Universal Robots PolyScope program: draw_test_name.urp

Program draw_test_name (installation=default directory=/programs createdIn=5.11.9.1010452 lastSavedIn=5.11.9.1010452 robotSerialNumber=20225200364)
Calibrated DH parameters: a=[0.00002, -0.569483, -0.54992, -0.00001, -0.000036, 0]; d=[0.180894, -146.691669, 192.918669, -46.053088, 0.119778, 0.115602]; alpha=[1.571425, -0.001534, 0.003359, 1.568739, -1.571477, 0]; deltaTheta=[0, 0.376258, -0.101074, -0.275185, -0.000002, 0]
Robot Program (runOnlyOnce=true)
  Script file /programs/usbdisk/draw_Marco_name.script
    | def Machining2():
    |   # Default parameters:
    |   global speed_ms = 0.3
    |   global speed_rads = 0.75
    |   global accel_mss = 3
    |   global accel_radss = 1.2
    |   global blend_radius_m = 0.001
    | 
    |   # Add subprograms here
    |   # Start of main program
    |   # Program generated by RoboDK v5.6.5 for UR10e on 20/10/2023 11:07:04
    |   # Using nominal kinematics.
    |   blend_radius_m = 0.001
    |   speed_ms = 1.000
    |   # set_reference(p[0.335000, -0.152000, -0.001000, 0.000000, 0.000000, 0.000000])
    |   set_tcp(p[0.000000, 0.000000, 0.252000, 0.000000, 0.000000, 0.000000])
    |   # Show Tool
    |   movej([0.142122, -1.120207, -2.573393, -1.018789, 1.570796, 1.712919],accel_radss,speed_rads,0,blend_radius_m)
    |   movel([0.142122, -1.120207, -2.573393, -1.018789, 1.570796, 1.712919],accel_mss,speed_ms,0,blend_radius_m)
    |   # Splitting Linear movement in 72 (instruction 7: MoveL 3)
    |   movel([0.142122, -1.121315, -2.574321, -1.016753, 1.570796, 1.712919],accel_mss,speed_ms,0,blend_radius_m)
    |   movel([0.142122, -1.122427, -2.575248, -1.014714, 1.570796, 1.712919],accel_mss,speed_ms,0,blend_radius_m)
    |   movel([0.142122, -1.123545, -2.576174, -1.012670, 1.570796, 1.712919],accel_mss,speed_ms,0,blend_radius_m)
    |   movel([0.142122, -1.124668, -2.577098, -1.010623, 1.570796, 1.712919],accel_mss,speed_ms,0,blend_radius_m)
    |   movel([0.142122, -1.125797, -2.578021, -1.008571, 1.570796, 1.712919],accel_mss,speed_ms,0,blend_radius_m)
    |   movel([0.142122, -1.126931, -2.578943, -1.006515, 1.570796, 1.712919],accel_mss,speed_ms,0,blend_radius_m)
    |   movel([0.142122, -1.128070, -2.579864, -1.004456, 1.570796, 1.712919],accel_mss,speed_ms,0,blend_radius_m)
    |   movel([0.142122, -1.129214, -2.580783, -1.002392, 1.570796, 1.712919],accel_mss,speed_ms,0,blend_radius_m)
    |   movel([0.142122, -1.130364, -2.581701, -1.000323, 1.570796, 1.712919],accel_mss,speed_ms,0,blend_radius_m)
    |   movel([0.142122, -1.131520, -2.582618, -0.998251, 1.570796, 1.712919],accel_mss,speed_ms,0,blend_radius_m)
    |   movel([0.142122, -1.132681, -2.583534, -0.996175, 1.570796, 1.712919],accel_mss,speed_ms,0,blend_radius_m)
    |   movel([0.142122, -1.133847, -2.584448, -0.994094, 1.570796, 1.712919],accel_mss,speed_ms,0,blend_radius_m)
    |   movel([0.142122, -1.135018, -2.585361, -0.992009, 1.570796, 1.712919],accel_mss,speed_ms,0,blend_radius_m)
    |   movel([0.142122, -1.136196, -2.586273, -0.989920, 1.570796, 1.712919],accel_mss,speed_ms,0,blend_radius_m)
    |   movel([0.142122, -1.137378, -2.587184, -0.987827, 1.570796, 1.712919],accel_mss,speed_ms,0,blend_radius_m)
    |   movel([0.142122, -1.138567, -2.588093, -0.985729, 1.570796, 1.712919],accel_mss,speed_ms,0,blend_radius_m)
    |   movel([0.142122, -1.139760, -2.589001, -0.983628, 1.570796, 1.712919],accel_mss,speed_ms,0,blend_radius_m)
    |   movel([0.142122, -1.140959, -2.589908, -0.981522, 1.570796, 1.712919],accel_mss,speed_ms,0,blend_radius_m)
    |   movel([0.142122, -1.142164, -2.590813, -0.979411, 1.570796, 1.712919],accel_mss,speed_ms,0,blend_radius_m)
    |   movel([0.142122, -1.143375, -2.591717, -0.977297, 1.570796, 1.712919],accel_mss,speed_ms,0,blend_radius_m)
    |   movel([0.142122, -1.144591, -2.592620, -0.975178, 1.570796, 1.712919],accel_mss,speed_ms,0,blend_radius_m)
    |   movel([0.142122, -1.145812, -2.593522, -0.973055, 1.570796, 1.712919],accel_mss,speed_ms,0,blend_radius_m)
    |   movel([0.142122, -1.147039, -2.594422, -0.970928, 1.570796, 1.712919],accel_mss,speed_ms,0,blend_radius_m)
    |   movel([0.142122, -1.148272, -2.595321, -0.968796, 1.570796, 1.712919],accel_mss,speed_ms,0,blend_radius_m)
    |   movel([0.142122, -1.149511, -2.596218, -0.966660, 1.570796, 1.712919],accel_mss,speed_ms,0,blend_radius_m)
    |   movel([0.142122, -1.150755, -2.597115, -0.964519, 1.570796, 1.712919],accel_mss,speed_ms,0,blend_radius_m)
    |   movel([0.142122, -1.152005, -2.598010, -0.962374, 1.570796, 1.712919],accel_mss,speed_ms,0,blend_radius_m)
    |   movel([0.142122, -1.153261, -2.598903, -0.960225, 1.570796, 1.712919],accel_mss,speed_ms,0,blend_radius_m)
    |   movel([0.142122, -1.154522, -2.599795, -0.958072, 1.570796, 1.712919],accel_mss,speed_ms,0,blend_radius_m)
    |   movel([0.142122, -1.155789, -2.600686, -0.955914, 1.570796, 1.712919],accel_mss,speed_ms,0,blend_radius_m)
    |   movel([0.142122, -1.157062, -2.601576, -0.953751, 1.570796, 1.712919],accel_mss,speed_ms,0,blend_radius_m)
    |   movel([0.142122, -1.158341, -2.602464, -0.951585, 1.570796, 1.712919],accel_mss,speed_ms,0,blend_radius_m)
    |   movel([0.142122, -1.159625, -2.603351, -0.949413, 1.570796, 1.712919],accel_mss,speed_ms,0,blend_radius_m)
    |   movel([0.142122, -1.160915, -2.604236, -0.947238, 1.570796, 1.712919],accel_mss,speed_ms,0,blend_radius_m)
    |   movel([0.142122, -1.162211, -2.605120, -0.945058, 1.570796, 1.712919],accel_mss,speed_ms,0,blend_radius_m)
    |   movel([0.142122, -1.163513, -2.606003, -0.942873, 1.570796, 1.712919],accel_mss,speed_ms,0,blend_radius_m)
    |   movel([0.142122, -1.164821, -2.606884, -0.940684, 1.570796, 1.712919],accel_mss,speed_ms,0,blend_radius_m)
    |   movel([0.142122, -1.166135, -2.607764, -0.938490, 1.570796, 1.712919],accel_mss,speed_ms,0,blend_radius_m)
    |   movel([0.142122, -1.167455, -2.608642, -0.936292, 1.570796, 1.712919],accel_mss,speed_ms,0,blend_radius_m)
    |   movel([0.142122, -1.168780, -2.609519, -0.934090, 1.570796, 1.712919],accel_mss,speed_ms,0,blend_radius_m)
    |   movel([0.142122, -1.170112, -2.610395, -0.931882, 1.570796, 1.712919],accel_mss,speed_ms,0,blend_radius_m)
    |   movel([0.142122, -1.171449, -2.611269, -0.929671, 1.570796, 1.712919],accel_mss,speed_ms,0,blend_radius_m)
    |   movel([0.142122, -1.172792, -2.612142, -0.927455, 1.570796, 1.712919],accel_mss,speed_ms,0,blend_radius_m)
    |   movel([0.142122, -1.174142, -2.613013, -0.925234, 1.570796, 1.712919],accel_mss,speed_ms,0,blend_radius_m)
    |   movel([0.142122, -1.175497, -2.613883, -0.923008, 1.570796, 1.712919],accel_mss,speed_ms,0,blend_radius_m)
    |   movel([0.142122, -1.176859, -2.614752, -0.920779, 1.570796, 1.712919],accel_mss,speed_ms,0,blend_radius_m)
    |   movel([0.142122, -1.178226, -2.615619, -0.918544, 1.570796, 1.712919],accel_mss,speed_ms,0,blend_radius_m)
    |   movel([0.142122, -1.179600, -2.616484, -0.916305, 1.570796, 1.712919],accel_mss,speed_ms,0,blend_radius_m)
    |   movel([0.142122, -1.180979, -2.617348, -0.914061, 1.570796, 1.712919],accel_mss,speed_ms,0,blend_radius_m)
    |   movel([0.142122, -1.182365, -2.618211, -0.911813, 1.570796, 1.712919],accel_mss,speed_ms,0,blend_radius_m)
    |   movel([0.142122, -1.183757, -2.619072, -0.909560, 1.570796, 1.712919],accel_mss,speed_ms,0,blend_radius_m)
    |   movel([0.142122, -1.185155, -2.619932, -0.907302, 1.570796, 1.712919],accel_mss,speed_ms,0,blend_radius_m)
    |   movel([0.142122, -1.186559, -2.620790, -0.905040, 1.570796, 1.712919],accel_mss,speed_ms,0,blend_radius_m)
    |   movel([0.142122, -1.187969, -2.621647, -0.902773, 1.570796, 1.712919],accel_mss,speed_ms,0,blend_radius_m)
    |   movel([0.142122, -1.189386, -2.622502, -0.900501, 1.570796, 1.712919],accel_mss,speed_ms,0,blend_radius_m)
    |   movel([0.142122, -1.190808, -2.623356, -0.898225, 1.570796, 1.712919],accel_mss,speed_ms,0,blend_radius_m)
    |   movel([0.142122, -1.192237, -2.624208, -0.895943, 1.570796, 1.712919],accel_mss,speed_ms,0,blend_radius_m)
    |   movel([0.142122, -1.193672, -2.625059, -0.893658, 1.570796, 1.712919],accel_mss,speed_ms,0,blend_radius_m)
    |   movel([0.142122, -1.195113, -2.625908, -0.891367, 1.570796, 1.712919],accel_mss,speed_ms,0,blend_radius_m)
    |   movel([0.142122, -1.196561, -2.626756, -0.889072, 1.570796, 1.712919],accel_mss,speed_ms,0,blend_radius_m)
    |   movel([0.142122, -1.198015, -2.627602, -0.886772, 1.570796, 1.712919],accel_mss,speed_ms,0,blend_radius_m)
    |   movel([0.142122, -1.199475, -2.628447, -0.884467, 1.570796, 1.712919],accel_mss,speed_ms,0,blend_radius_m)
    |   movel([0.142122, -1.200942, -2.629290, -0.882157, 1.570796, 1.712919],accel_mss,speed_ms,0,blend_radius_m)
    |   movel([0.142122, -1.202414, -2.630132, -0.879843, 1.570796, 1.712919],accel_mss,speed_ms,0,blend_radius_m)
    |   movel([0.142122, -1.203893, -2.630972, -0.877524, 1.570796, 1.712919],accel_mss,speed_ms,0,blend_radius_m)
    |   movel([0.142122, -1.205379, -2.631810, -0.875200, 1.570796, 1.712919],accel_mss,speed_ms,0,blend_radius_m)
    |   movel([0.142122, -1.206871, -2.632647, -0.872871, 1.570796, 1.712919],accel_mss,speed_ms,0,blend_radius_m)
    |   movel([0.142122, -1.208369, -2.633482, -0.870538, 1.570796, 1.712919],accel_mss,speed_ms,0,blend_radius_m)
    |   movel([0.142122, -1.209874, -2.634316, -0.868199, 1.570796, 1.712919],accel_mss,speed_ms,0,blend_radius_m)
    |   movel([0.142122, -1.211385, -2.635148, -0.865856, 1.570796, 1.712919],accel_mss,speed_ms,0,blend_radius_m)
    |   movel([0.142122, -1.212902, -2.635979, -0.863508, 1.570796, 1.712919],accel_mss,speed_ms,0,blend_radius_m)
    |   movel([0.142122, -1.214426, -2.636807, -0.861155, 1.570796, 1.712919],accel_mss,speed_ms,0,blend_radius_m)
    |   movel([0.142122, -1.214426, -2.636807, -0.861155, 1.570796, 1.712919],accel_mss,speed_ms,0,blend_radius_m)
    |   speed_ms = 1.000
    |   # Splitting Linear movement in 8 (instruction 10: MoveL 5)
    |   movel([0.142122, -1.215804, -2.637552, -0.859033, 1.570796, 1.712919],accel_mss,speed_ms,0,blend_radius_m)
    |   movel([0.142122, -1.217186, -2.638295, -0.856907, 1.570796, 1.712919],accel_mss,speed_ms,0,blend_radius_m)
    |   movel([0.142122, -1.218574, -2.639038, -0.854778, 1.570796, 1.712919],accel_mss,speed_ms,0,blend_radius_m)
    |   movel([0.142122, -1.219967, -2.639778, -0.852644, 1.570796, 1.712919],accel_mss,speed_ms,0,blend_radius_m)
    |   movel([0.142122, -1.221365, -2.640518, -0.850506, 1.570796, 1.712919],accel_mss,speed_ms,0,blend_radius_m)
    |   movel([0.142122, -1.222769, -2.641256, -0.848365, 1.570796, 1.712919],accel_mss,speed_ms,0,blend_radius_m)
    |   movel([0.142122, -1.224177, -2.641992, -0.846219, 1.570796, 1.712919],accel_mss,speed_ms,0,blend_radius_m)
    |   movel([0.142122, -1.225592, -2.642728, -0.844069, 1.570796, 1.712919],accel_mss,speed_ms,0,blend_radius_m)
    |   movel([0.142122, -1.225592, -2.642728, -0.844069, 1.570796, 1.712919],accel_mss,speed_ms,0,blend_radius_m)
    |   # Splitting Linear movement in 16 (instruction 12: MoveL 7)
    |   movel([0.142122, -1.227011, -2.643462, -0.841916, 1.570796, 1.712919],accel_mss,speed_ms,0,blend_radius_m)
    |   movel([0.142122, -1.228436, -2.644195, -0.839758, 1.570796, 1.712919],accel_mss,speed_ms,0,blend_radius_m)
    |   movel([0.142122, -1.229866, -2.644926, -0.837597, 1.570796, 1.712919],accel_mss,speed_ms,0,blend_radius_m)
    |   movel([0.142122, -1.231302, -2.645656, -0.835431, 1.570796, 1.712919],accel_mss,speed_ms,0,blend_radius_m)
    |   movel([0.142122, -1.232743, -2.646385, -0.833261, 1.570796, 1.712919],accel_mss,speed_ms,0,blend_radius_m)
    |   movel([0.142122, -1.234189, -2.647112, -0.831088, 1.570796, 1.712919],accel_mss,speed_ms,0,blend_radius_m)
    |   movel([0.142122, -1.235641, -2.647838, -0.828910, 1.570796, 1.712919],accel_mss,speed_ms,0,blend_radius_m)
    |   movel([0.142122, -1.237099, -2.648562, -0.826728, 1.570796, 1.712919],accel_mss,speed_ms,0,blend_radius_m)
    |   movel([0.142122, -1.238561, -2.649286, -0.824542, 1.570796, 1.712919],accel_mss,speed_ms,0,blend_radius_m)
    |   movel([0.142122, -1.240029, -2.650007, -0.822352, 1.570796, 1.712919],accel_mss,speed_ms,0,blend_radius_m)
    |   movel([0.142122, -1.241503, -2.650728, -0.820158, 1.570796, 1.712919],accel_mss,speed_ms,0,blend_radius_m)
    |   movel([0.142122, -1.242982, -2.651447, -0.817960, 1.570796, 1.712919],accel_mss,speed_ms,0,blend_radius_m)
    |   movel([0.142122, -1.244466, -2.652164, -0.815758, 1.570796, 1.712919],accel_mss,speed_ms,0,blend_radius_m)
    |   movel([0.142122, -1.245956, -2.652880, -0.813552, 1.570796, 1.712919],accel_mss,speed_ms,0,blend_radius_m)
    |   movel([0.142122, -1.247452, -2.653595, -0.811342, 1.570796, 1.712919],accel_mss,speed_ms,0,blend_radius_m)
    |   movel([0.142122, -1.248953, -2.654308, -0.809128, 1.570796, 1.712919],accel_mss,speed_ms,0,blend_radius_m)
    |   # Splitting Linear movement in 6 (instruction 13: MoveL 8)
    |   movel([0.140118, -1.249589, -2.653970, -0.808830, 1.570796, 1.710915],accel_mss,speed_ms,0,blend_radius_m)
    |   movel([0.138115, -1.250228, -2.653630, -0.808531, 1.570796, 1.708912],accel_mss,speed_ms,0,blend_radius_m)
    |   movel([0.136113, -1.250869, -2.653288, -0.808232, 1.570796, 1.706910],accel_mss,speed_ms,0,blend_radius_m)
    |   movel([0.134112, -1.251512, -2.652944, -0.807932, 1.570796, 1.704909],accel_mss,speed_ms,0,blend_radius_m)
    |   movel([0.132112, -1.252158, -2.652599, -0.807632, 1.570796, 1.702908],accel_mss,speed_ms,0,blend_radius_m)
    |   movel([0.130113, -1.252807, -2.652252, -0.807331, 1.570796, 1.700909],accel_mss,speed_ms,0,blend_radius_m)
    |   # Splitting Linear movement in 16 (instruction 14: MoveL 9)
    |   movel([0.130113, -1.251309, -2.651541, -0.809539, 1.570796, 1.700909],accel_mss,speed_ms,0,blend_radius_m)
    |   movel([0.130113, -1.249816, -2.650829, -0.811744, 1.570796, 1.700909],accel_mss,speed_ms,0,blend_radius_m)
    |   movel([0.130113, -1.248329, -2.650116, -0.813944, 1.570796, 1.700909],accel_mss,speed_ms,0,blend_radius_m)
    |   movel([0.130113, -1.246847, -2.649401, -0.816141, 1.570796, 1.700909],accel_mss,speed_ms,0,blend_radius_m)
    |   movel([0.130113, -1.245371, -2.648685, -0.818333, 1.570796, 1.700909],accel_mss,speed_ms,0,blend_radius_m)
    |   movel([0.130113, -1.243900, -2.647967, -0.820522, 1.570796, 1.700909],accel_mss,speed_ms,0,blend_radius_m)
    |   movel([0.130113, -1.242435, -2.647248, -0.822706, 1.570796, 1.700909],accel_mss,speed_ms,0,blend_radius_m)
    |   movel([0.130113, -1.240974, -2.646528, -0.824887, 1.570796, 1.700909],accel_mss,speed_ms,0,blend_radius_m)
    |   movel([0.130113, -1.239520, -2.645806, -0.827063, 1.570796, 1.700909],accel_mss,speed_ms,0,blend_radius_m)
    |   movel([0.130113, -1.238071, -2.645083, -0.829236, 1.570796, 1.700909],accel_mss,speed_ms,0,blend_radius_m)
    |   movel([0.130113, -1.236627, -2.644358, -0.831404, 1.570796, 1.700909],accel_mss,speed_ms,0,blend_radius_m)
    |   movel([0.130113, -1.235188, -2.643632, -0.833569, 1.570796, 1.700909],accel_mss,speed_ms,0,blend_radius_m)
    |   movel([0.130113, -1.233755, -2.642905, -0.835729, 1.570796, 1.700909],accel_mss,speed_ms,0,blend_radius_m)
    |   movel([0.130113, -1.232327, -2.642176, -0.837886, 1.570796, 1.700909],accel_mss,speed_ms,0,blend_radius_m)
    |   movel([0.130113, -1.230904, -2.641446, -0.840038, 1.570796, 1.700909],accel_mss,speed_ms,0,blend_radius_m)
    |   movel([0.130113, -1.229487, -2.640715, -0.842187, 1.570796, 1.700909],accel_mss,speed_ms,0,blend_radius_m)
    |   # Splitting Linear movement in 6 (instruction 15: MoveL 10)
    |   movel([0.132112, -1.228832, -2.641055, -0.842503, 1.570796, 1.702908],accel_mss,speed_ms,0,blend_radius_m)
    |   movel([0.134112, -1.228179, -2.641393, -0.842817, 1.570796, 1.704909],accel_mss,speed_ms,0,blend_radius_m)
    |   movel([0.136113, -1.227528, -2.641729, -0.843131, 1.570796, 1.706910],accel_mss,speed_ms,0,blend_radius_m)
    |   movel([0.138115, -1.226880, -2.642064, -0.843445, 1.570796, 1.708912],accel_mss,speed_ms,0,blend_radius_m)
    |   movel([0.140118, -1.226235, -2.642397, -0.843758, 1.570796, 1.710915],accel_mss,speed_ms,0,blend_radius_m)
    |   movel([0.142122, -1.225592, -2.642728, -0.844069, 1.570796, 1.712919],accel_mss,speed_ms,0,blend_radius_m)
    |   # Splitting Linear movement in 16 (instruction 16: MoveL 11)
    |   movel([0.142122, -1.227011, -2.643462, -0.841916, 1.570796, 1.712919],accel_mss,speed_ms,0,blend_radius_m)
    |   movel([0.142122, -1.228436, -2.644195, -0.839758, 1.570796, 1.712919],accel_mss,speed_ms,0,blend_radius_m)
    |   movel([0.142122, -1.229866, -2.644926, -0.837597, 1.570796, 1.712919],accel_mss,speed_ms,0,blend_radius_m)
    |   movel([0.142122, -1.231302, -2.645656, -0.835431, 1.570796, 1.712919],accel_mss,speed_ms,0,blend_radius_m)
    |   movel([0.142122, -1.232743, -2.646385, -0.833261, 1.570796, 1.712919],accel_mss,speed_ms,0,blend_radius_m)
    |   movel([0.142122, -1.234189, -2.647112, -0.831088, 1.570796, 1.712919],accel_mss,speed_ms,0,blend_radius_m)
    |   movel([0.142122, -1.235641, -2.647838, -0.828910, 1.570796, 1.712919],accel_mss,speed_ms,0,blend_radius_m)
    |   movel([0.142122, -1.237099, -2.648562, -0.826728, 1.570796, 1.712919],accel_mss,speed_ms,0,blend_radius_m)
    |   movel([0.142122, -1.238561, -2.649286, -0.824542, 1.570796, 1.712919],accel_mss,speed_ms,0,blend_radius_m)
    |   movel([0.142122, -1.240029, -2.650007, -0.822352, 1.570796, 1.712919],accel_mss,speed_ms,0,blend_radius_m)
    |   movel([0.142122, -1.241503, -2.650728, -0.820158, 1.570796, 1.712919],accel_mss,speed_ms,0,blend_radius_m)
    |   movel([0.142122, -1.242982, -2.651447, -0.817960, 1.570796, 1.712919],accel_mss,speed_ms,0,blend_radius_m)
    |   movel([0.142122, -1.244466, -2.652164, -0.815758, 1.570796, 1.712919],accel_mss,speed_ms,0,blend_radius_m)
    |   movel([0.142122, -1.245956, -2.652880, -0.813552, 1.570796, 1.712919],accel_mss,speed_ms,0,blend_radius_m)
    |   movel([0.142122, -1.247452, -2.653595, -0.811342, 1.570796, 1.712919],accel_mss,speed_ms,0,blend_radius_m)
    |   movel([0.142122, -1.248953, -2.654308, -0.809128, 1.570796, 1.712919],accel_mss,speed_ms,0,blend_radius_m)
    |   # Splitting Linear movement in 8 (instruction 17: MoveL 12)
    |   movel([0.140538, -1.249956, -2.653775, -0.808658, 1.570796, 1.711335],accel_mss,speed_ms,0,blend_radius_m)
    |   movel([0.138957, -1.250958, -2.653241, -0.808191, 1.570796, 1.709753],accel_mss,speed_ms,0,blend_radius_m)
    |   movel([0.137378, -1.251960, -2.652705, -0.807724, 1.570796, 1.708174],accel_mss,speed_ms,0,blend_radius_m)
    |   movel([0.135801, -1.252961, -2.652169, -0.807259, 1.570796, 1.706597],accel_mss,speed_ms,0,blend_radius_m)
    |   movel([0.134226, -1.253962, -2.651632, -0.806795, 1.570796, 1.705023],accel_mss,speed_ms,0,blend_radius_m)
    |   movel([0.132655, -1.254963, -2.651093, -0.806333, 1.570796, 1.703451],accel_mss,speed_ms,0,blend_radius_m)
    |   movel([0.131085, -1.255963, -2.650554, -0.805872, 1.570796, 1.701881],accel_mss,speed_ms,0,blend_radius_m)
    |   movel([0.129518, -1.256963, -2.650014, -0.805412, 1.570796, 1.700314],accel_mss,speed_ms,0,blend_radius_m)
    |   # Splitting Linear movement in 16 (instruction 18: MoveL 13)
    |   movel([0.129518, -1.255469, -2.649306, -0.807614, 1.570796, 1.700314],accel_mss,speed_ms,0,blend_radius_m)
    |   movel([0.129518, -1.253979, -2.648597, -0.809813, 1.570796, 1.700314],accel_mss,speed_ms,0,blend_radius_m)
    |   movel([0.129518, -1.252495, -2.647887, -0.812007, 1.570796, 1.700314],accel_mss,speed_ms,0,blend_radius_m)
    |   movel([0.129518, -1.251017, -2.647175, -0.814198, 1.570796, 1.700314],accel_mss,speed_ms,0,blend_radius_m)
    |   movel([0.129518, -1.249543, -2.646461, -0.816384, 1.570796, 1.700314],accel_mss,speed_ms,0,blend_radius_m)
    |   movel([0.129518, -1.248076, -2.645747, -0.818567, 1.570796, 1.700314],accel_mss,speed_ms,0,blend_radius_m)
    |   movel([0.129518, -1.246613, -2.645031, -0.820745, 1.570796, 1.700314],accel_mss,speed_ms,0,blend_radius_m)
    |   movel([0.129518, -1.245156, -2.644313, -0.822920, 1.570796, 1.700314],accel_mss,speed_ms,0,blend_radius_m)
    |   movel([0.129518, -1.243704, -2.643594, -0.825091, 1.570796, 1.700314],accel_mss,speed_ms,0,blend_radius_m)
    |   movel([0.129518, -1.242257, -2.642874, -0.827257, 1.570796, 1.700314],accel_mss,speed_ms,0,blend_radius_m)
    |   movel([0.129518, -1.240816, -2.642152, -0.829420, 1.570796, 1.700314],accel_mss,speed_ms,0,blend_radius_m)
    |   movel([0.129518, -1.239380, -2.641429, -0.831579, 1.570796, 1.700314],accel_mss,speed_ms,0,blend_radius_m)
    |   movel([0.129518, -1.237950, -2.640705, -0.833734, 1.570796, 1.700314],accel_mss,speed_ms,0,blend_radius_m)
    |   movel([0.129518, -1.236524, -2.639979, -0.835885, 1.570796, 1.700314],accel_mss,speed_ms,0,blend_radius_m)
    |   movel([0.129518, -1.235104, -2.639252, -0.838032, 1.570796, 1.700314],accel_mss,speed_ms,0,blend_radius_m)
    |   movel([0.129518, -1.233690, -2.638524, -0.840176, 1.570796, 1.700314],accel_mss,speed_ms,0,blend_radius_m)
    |   # Splitting Linear movement in 8 (instruction 19: MoveL 14)
    |   movel([0.130935, -1.233727, -2.638504, -0.840158, 1.570796, 1.701732],accel_mss,speed_ms,0,blend_radius_m)
    |   movel([0.132351, -1.233767, -2.638483, -0.840139, 1.570796, 1.703148],accel_mss,speed_ms,0,blend_radius_m)
    |   movel([0.133766, -1.233809, -2.638461, -0.840119, 1.570796, 1.704563],accel_mss,speed_ms,0,blend_radius_m)
    |   movel([0.135180, -1.233853, -2.638438, -0.840098, 1.570796, 1.705976],accel_mss,speed_ms,0,blend_radius_m)
    |   movel([0.136593, -1.233900, -2.638414, -0.840075, 1.570796, 1.707389],accel_mss,speed_ms,0,blend_radius_m)
    |   movel([0.138004, -1.233949, -2.638388, -0.840052, 1.570796, 1.708800],accel_mss,speed_ms,0,blend_radius_m)
    |   movel([0.139414, -1.234000, -2.638361, -0.840028, 1.570796, 1.710211],accel_mss,speed_ms,0,blend_radius_m)
    |   movel([0.140824, -1.234053, -2.638333, -0.840003, 1.570796, 1.711620],accel_mss,speed_ms,0,blend_radius_m)
    |   # Splitting Linear movement in 16 (instruction 20: MoveL 15)
    |   movel([0.140824, -1.235468, -2.639062, -0.837860, 1.570796, 1.711620],accel_mss,speed_ms,0,blend_radius_m)
    |   movel([0.140824, -1.236888, -2.639788, -0.835713, 1.570796, 1.711620],accel_mss,speed_ms,0,blend_radius_m)
    |   movel([0.140824, -1.238313, -2.640514, -0.833563, 1.570796, 1.711620],accel_mss,speed_ms,0,blend_radius_m)
    |   movel([0.140824, -1.239743, -2.641238, -0.831408, 1.570796, 1.711620],accel_mss,speed_ms,0,blend_radius_m)
    |   movel([0.140824, -1.241179, -2.641961, -0.829250, 1.570796, 1.711620],accel_mss,speed_ms,0,blend_radius_m)
    |   movel([0.140824, -1.242620, -2.642682, -0.827087, 1.570796, 1.711620],accel_mss,speed_ms,0,blend_radius_m)
    |   movel([0.140824, -1.244066, -2.643402, -0.824921, 1.570796, 1.711620],accel_mss,speed_ms,0,blend_radius_m)
    |   movel([0.140824, -1.245518, -2.644121, -0.822751, 1.570796, 1.711620],accel_mss,speed_ms,0,blend_radius_m)
    |   movel([0.140824, -1.246974, -2.644838, -0.820577, 1.570796, 1.711620],accel_mss,speed_ms,0,blend_radius_m)
    |   movel([0.140824, -1.248437, -2.645554, -0.818399, 1.570796, 1.711620],accel_mss,speed_ms,0,blend_radius_m)
    |   movel([0.140824, -1.249904, -2.646268, -0.816217, 1.570796, 1.711620],accel_mss,speed_ms,0,blend_radius_m)
    |   movel([0.140824, -1.251377, -2.646981, -0.814031, 1.570796, 1.711620],accel_mss,speed_ms,0,blend_radius_m)
    |   movel([0.140824, -1.252856, -2.647693, -0.811841, 1.570796, 1.711620],accel_mss,speed_ms,0,blend_radius_m)
    |   movel([0.140824, -1.254339, -2.648403, -0.809647, 1.570796, 1.711620],accel_mss,speed_ms,0,blend_radius_m)
    |   movel([0.140824, -1.255828, -2.649112, -0.807449, 1.570796, 1.711620],accel_mss,speed_ms,0,blend_radius_m)
    |   movel([0.140824, -1.257323, -2.649819, -0.805247, 1.570796, 1.711620],accel_mss,speed_ms,0,blend_radius_m)
    |   # Splitting Linear movement in 8 (instruction 21: MoveL 16)
    |   movel([0.139414, -1.257270, -2.649847, -0.805271, 1.570796, 1.710211],accel_mss,speed_ms,0,blend_radius_m)
    |   movel([0.138004, -1.257220, -2.649875, -0.805294, 1.570796, 1.708800],accel_mss,speed_ms,0,blend_radius_m)
    |   movel([0.136593, -1.257171, -2.649901, -0.805317, 1.570796, 1.707389],accel_mss,speed_ms,0,blend_radius_m)
    |   movel([0.135180, -1.257125, -2.649926, -0.805338, 1.570796, 1.705976],accel_mss,speed_ms,0,blend_radius_m)
    |   movel([0.133766, -1.257082, -2.649950, -0.805358, 1.570796, 1.704563],accel_mss,speed_ms,0,blend_radius_m)
    |   movel([0.132351, -1.257040, -2.649972, -0.805377, 1.570796, 1.703148],accel_mss,speed_ms,0,blend_radius_m)
    |   movel([0.130935, -1.257001, -2.649993, -0.805395, 1.570796, 1.701732],accel_mss,speed_ms,0,blend_radius_m)
    |   movel([0.129518, -1.256963, -2.650014, -0.805412, 1.570796, 1.700314],accel_mss,speed_ms,0,blend_radius_m)
    |   # Splitting Linear movement in 16 (instruction 22: MoveL 17)
    |   movel([0.129518, -1.255469, -2.649306, -0.807614, 1.570796, 1.700314],accel_mss,speed_ms,0,blend_radius_m)
    |   movel([0.129518, -1.253979, -2.648597, -0.809813, 1.570796, 1.700314],accel_mss,speed_ms,0,blend_radius_m)
    |   movel([0.129518, -1.252495, -2.647887, -0.812007, 1.570796, 1.700314],accel_mss,speed_ms,0,blend_radius_m)
    |   movel([0.129518, -1.251017, -2.647175, -0.814198, 1.570796, 1.700314],accel_mss,speed_ms,0,blend_radius_m)
    |   movel([0.129518, -1.249543, -2.646461, -0.816384, 1.570796, 1.700314],accel_mss,speed_ms,0,blend_radius_m)
    |   movel([0.129518, -1.248076, -2.645747, -0.818567, 1.570796, 1.700314],accel_mss,speed_ms,0,blend_radius_m)
    |   movel([0.129518, -1.246613, -2.645031, -0.820745, 1.570796, 1.700314],accel_mss,speed_ms,0,blend_radius_m)
    |   movel([0.129518, -1.245156, -2.644313, -0.822920, 1.570796, 1.700314],accel_mss,speed_ms,0,blend_radius_m)
    |   movel([0.129518, -1.243704, -2.643594, -0.825091, 1.570796, 1.700314],accel_mss,speed_ms,0,blend_radius_m)
    |   movel([0.129518, -1.242257, -2.642874, -0.827257, 1.570796, 1.700314],accel_mss,speed_ms,0,blend_radius_m)
    |   movel([0.129518, -1.240816, -2.642152, -0.829420, 1.570796, 1.700314],accel_mss,speed_ms,0,blend_radius_m)
    |   movel([0.129518, -1.239380, -2.641429, -0.831579, 1.570796, 1.700314],accel_mss,speed_ms,0,blend_radius_m)
    |   movel([0.129518, -1.237950, -2.640705, -0.833734, 1.570796, 1.700314],accel_mss,speed_ms,0,blend_radius_m)
    |   movel([0.129518, -1.236524, -2.639979, -0.835885, 1.570796, 1.700314],accel_mss,speed_ms,0,blend_radius_m)
    |   movel([0.129518, -1.235104, -2.639252, -0.838032, 1.570796, 1.700314],accel_mss,speed_ms,0,blend_radius_m)
    |   movel([0.129518, -1.233690, -2.638524, -0.840176, 1.570796, 1.700314],accel_mss,speed_ms,0,blend_radius_m)
    |   # Splitting Linear movement in 8 (instruction 23: MoveL 18)
    |   movel([0.130935, -1.233727, -2.638504, -0.840158, 1.570796, 1.701732],accel_mss,speed_ms,0,blend_radius_m)
    |   movel([0.132351, -1.233767, -2.638483, -0.840139, 1.570796, 1.703148],accel_mss,speed_ms,0,blend_radius_m)
    |   movel([0.133766, -1.233809, -2.638461, -0.840119, 1.570796, 1.704563],accel_mss,speed_ms,0,blend_radius_m)
    |   movel([0.135180, -1.233853, -2.638438, -0.840098, 1.570796, 1.705976],accel_mss,speed_ms,0,blend_radius_m)
    |   movel([0.136593, -1.233900, -2.638414, -0.840075, 1.570796, 1.707389],accel_mss,speed_ms,0,blend_radius_m)
    |   movel([0.138004, -1.233949, -2.638388, -0.840052, 1.570796, 1.708800],accel_mss,speed_ms,0,blend_radius_m)
    |   movel([0.139414, -1.234000, -2.638361, -0.840028, 1.570796, 1.710211],accel_mss,speed_ms,0,blend_radius_m)
    |   movel([0.140824, -1.234053, -2.638333, -0.840003, 1.570796, 1.711620],accel_mss,speed_ms,0,blend_radius_m)
    |   # Splitting Linear movement in 16 (instruction 24: MoveL 19)
    |   movel([0.140824, -1.235468, -2.639062, -0.837860, 1.570796, 1.711620],accel_mss,speed_ms,0,blend_radius_m)
    |   movel([0.140824, -1.236888, -2.639788, -0.835713, 1.570796, 1.711620],accel_mss,speed_ms,0,blend_radius_m)
    |   movel([0.140824, -1.238313, -2.640514, -0.833563, 1.570796, 1.711620],accel_mss,speed_ms,0,blend_radius_m)
    |   movel([0.140824, -1.239743, -2.641238, -0.831408, 1.570796, 1.711620],accel_mss,speed_ms,0,blend_radius_m)
    |   movel([0.140824, -1.241179, -2.641961, -0.829250, 1.570796, 1.711620],accel_mss,speed_ms,0,blend_radius_m)
    |   movel([0.140824, -1.242620, -2.642682, -0.827087, 1.570796, 1.711620],accel_mss,speed_ms,0,blend_radius_m)
    |   movel([0.140824, -1.244066, -2.643402, -0.824921, 1.570796, 1.711620],accel_mss,speed_ms,0,blend_radius_m)
    |   movel([0.140824, -1.245518, -2.644121, -0.822751, 1.570796, 1.711620],accel_mss,speed_ms,0,blend_radius_m)
    |   movel([0.140824, -1.246974, -2.644838, -0.820577, 1.570796, 1.711620],accel_mss,speed_ms,0,blend_radius_m)
    |   movel([0.140824, -1.248437, -2.645554, -0.818399, 1.570796, 1.711620],accel_mss,speed_ms,0,blend_radius_m)
    |   movel([0.140824, -1.249904, -2.646268, -0.816217, 1.570796, 1.711620],accel_mss,speed_ms,0,blend_radius_m)
    |   movel([0.140824, -1.251377, -2.646981, -0.814031, 1.570796, 1.711620],accel_mss,speed_ms,0,blend_radius_m)
    |   movel([0.140824, -1.252856, -2.647693, -0.811841, 1.570796, 1.711620],accel_mss,speed_ms,0,blend_radius_m)
    |   movel([0.140824, -1.254339, -2.648403, -0.809647, 1.570796, 1.711620],accel_mss,speed_ms,0,blend_radius_m)
    |   movel([0.140824, -1.255828, -2.649112, -0.807449, 1.570796, 1.711620],accel_mss,speed_ms,0,blend_radius_m)
    |   movel([0.140824, -1.257323, -2.649819, -0.805247, 1.570796, 1.711620],accel_mss,speed_ms,0,blend_radius_m)
    |   # Splitting Linear movement in 6 (instruction 25: MoveL 20)
    |   movel([0.138839, -1.257945, -2.649482, -0.804962, 1.570796, 1.709635],accel_mss,speed_ms,0,blend_radius_m)
    |   movel([0.136855, -1.258570, -2.649143, -0.804676, 1.570796, 1.707651],accel_mss,speed_ms,0,blend_radius_m)
    |   movel([0.134872, -1.259197, -2.648802, -0.804390, 1.570796, 1.705668],accel_mss,speed_ms,0,blend_radius_m)
    |   movel([0.132890, -1.259827, -2.648459, -0.804103, 1.570796, 1.703686],accel_mss,speed_ms,0,blend_radius_m)
    |   movel([0.130909, -1.260459, -2.648115, -0.803815, 1.570796, 1.701705],accel_mss,speed_ms,0,blend_radius_m)
    |   movel([0.128929, -1.261093, -2.647769, -0.803527, 1.570796, 1.699725],accel_mss,speed_ms,0,blend_radius_m)
    |   # Splitting Linear movement in 16 (instruction 26: MoveL 21)
    |   movel([0.128929, -1.259602, -2.647064, -0.805723, 1.570796, 1.699725],accel_mss,speed_ms,0,blend_radius_m)
    |   movel([0.128929, -1.258116, -2.646358, -0.807915, 1.570796, 1.699725],accel_mss,speed_ms,0,blend_radius_m)
    |   movel([0.128929, -1.256635, -2.645651, -0.810103, 1.570796, 1.699725],accel_mss,speed_ms,0,blend_radius_m)
    |   movel([0.128929, -1.255159, -2.644942, -0.812288, 1.570796, 1.699725],accel_mss,speed_ms,0,blend_radius_m)
    |   movel([0.128929, -1.253689, -2.644231, -0.814468, 1.570796, 1.699725],accel_mss,speed_ms,0,blend_radius_m)
    |   movel([0.128929, -1.252224, -2.643520, -0.816645, 1.570796, 1.699725],accel_mss,speed_ms,0,blend_radius_m)
    |   movel([0.128929, -1.250765, -2.642807, -0.818817, 1.570796, 1.699725],accel_mss,speed_ms,0,blend_radius_m)
    |   movel([0.128929, -1.249311, -2.642092, -0.820986, 1.570796, 1.699725],accel_mss,speed_ms,0,blend_radius_m)
    |   movel([0.128929, -1.247862, -2.641376, -0.823151, 1.570796, 1.699725],accel_mss,speed_ms,0,blend_radius_m)
    |   movel([0.128929, -1.246418, -2.640659, -0.825312, 1.570796, 1.699725],accel_mss,speed_ms,0,blend_radius_m)
    |   movel([0.128929, -1.244980, -2.639940, -0.827469, 1.570796, 1.699725],accel_mss,speed_ms,0,blend_radius_m)
    |   movel([0.128929, -1.243546, -2.639220, -0.829622, 1.570796, 1.699725],accel_mss,speed_ms,0,blend_radius_m)
    |   movel([0.128929, -1.242119, -2.638499, -0.831772, 1.570796, 1.699725],accel_mss,speed_ms,0,blend_radius_m)
    |   movel([0.128929, -1.240696, -2.637776, -0.833917, 1.570796, 1.699725],accel_mss,speed_ms,0,blend_radius_m)
    |   movel([0.128929, -1.239278, -2.637052, -0.836059, 1.570796, 1.699725],accel_mss,speed_ms,0,blend_radius_m)
    |   movel([0.128929, -1.237866, -2.636326, -0.838197, 1.570796, 1.699725],accel_mss,speed_ms,0,blend_radius_m)
    |   # Splitting Linear movement in 8 (instruction 27: MoveL 22)
    |   movel([0.130293, -1.238231, -2.636133, -0.838025, 1.570796, 1.701089],accel_mss,speed_ms,0,blend_radius_m)
    |   movel([0.131656, -1.238598, -2.635939, -0.837852, 1.570796, 1.702452],accel_mss,speed_ms,0,blend_radius_m)
    |   movel([0.133016, -1.238967, -2.635743, -0.837679, 1.570796, 1.703812],accel_mss,speed_ms,0,blend_radius_m)
    |   movel([0.134374, -1.239339, -2.635546, -0.837504, 1.570796, 1.705170],accel_mss,speed_ms,0,blend_radius_m)
    |   movel([0.135730, -1.239713, -2.635348, -0.837328, 1.570796, 1.706527],accel_mss,speed_ms,0,blend_radius_m)
    |   movel([0.137084, -1.240089, -2.635148, -0.837152, 1.570796, 1.707881],accel_mss,speed_ms,0,blend_radius_m)
    |   movel([0.138436, -1.240468, -2.634947, -0.836974, 1.570796, 1.709233],accel_mss,speed_ms,0,blend_radius_m)
    |   movel([0.139786, -1.240849, -2.634744, -0.836796, 1.570796, 1.710582],accel_mss,speed_ms,0,blend_radius_m)
    |   # Splitting Linear movement in 16 (instruction 28: MoveL 23)
    |   movel([0.139786, -1.242259, -2.635467, -0.834662, 1.570796, 1.710582],accel_mss,speed_ms,0,blend_radius_m)
    |   movel([0.139786, -1.243675, -2.636189, -0.832524, 1.570796, 1.710582],accel_mss,speed_ms,0,blend_radius_m)
    |   movel([0.139786, -1.245096, -2.636910, -0.830383, 1.570796, 1.710582],accel_mss,speed_ms,0,blend_radius_m)
    |   movel([0.139786, -1.246522, -2.637630, -0.828238, 1.570796, 1.710582],accel_mss,speed_ms,0,blend_radius_m)
    |   movel([0.139786, -1.247953, -2.638348, -0.826088, 1.570796, 1.710582],accel_mss,speed_ms,0,blend_radius_m)
    |   movel([0.139786, -1.249389, -2.639064, -0.823935, 1.570796, 1.710582],accel_mss,speed_ms,0,blend_radius_m)
    |   movel([0.139786, -1.250831, -2.639779, -0.821778, 1.570796, 1.710582],accel_mss,speed_ms,0,blend_radius_m)
    |   movel([0.139786, -1.252278, -2.640493, -0.819618, 1.570796, 1.710582],accel_mss,speed_ms,0,blend_radius_m)
    |   movel([0.139786, -1.253730, -2.641206, -0.817453, 1.570796, 1.710582],accel_mss,speed_ms,0,blend_radius_m)
    |   movel([0.139786, -1.255187, -2.641917, -0.815285, 1.570796, 1.710582],accel_mss,speed_ms,0,blend_radius_m)
    |   movel([0.139786, -1.256650, -2.642626, -0.813113, 1.570796, 1.710582],accel_mss,speed_ms,0,blend_radius_m)
    |   movel([0.139786, -1.258118, -2.643335, -0.810936, 1.570796, 1.710582],accel_mss,speed_ms,0,blend_radius_m)
    |   movel([0.139786, -1.259591, -2.644041, -0.808756, 1.570796, 1.710582],accel_mss,speed_ms,0,blend_radius_m)
    |   movel([0.139786, -1.261070, -2.644747, -0.806573, 1.570796, 1.710582],accel_mss,speed_ms,0,blend_radius_m)
    |   movel([0.139786, -1.262553, -2.645451, -0.804385, 1.570796, 1.710582],accel_mss,speed_ms,0,blend_radius_m)
    |   movel([0.139786, -1.264042, -2.646153, -0.802193, 1.570796, 1.710582],accel_mss,speed_ms,0,blend_radius_m)
    |   # Splitting Linear movement in 8 (instruction 29: MoveL 24)
    |   movel([0.138387, -1.263987, -2.646184, -0.802218, 1.570796, 1.709184],accel_mss,speed_ms,0,blend_radius_m)
    |   movel([0.136987, -1.263934, -2.646213, -0.802242, 1.570796, 1.707784],accel_mss,speed_ms,0,blend_radius_m)
    |   movel([0.135586, -1.263883, -2.646241, -0.802265, 1.570796, 1.706382],accel_mss,speed_ms,0,blend_radius_m)
    |   movel([0.134184, -1.263834, -2.646268, -0.802287, 1.570796, 1.704980],accel_mss,speed_ms,0,blend_radius_m)
    |   movel([0.132780, -1.263788, -2.646293, -0.802308, 1.570796, 1.703577],accel_mss,speed_ms,0,blend_radius_m)
    |   movel([0.131376, -1.263743, -2.646318, -0.802328, 1.570796, 1.702172],accel_mss,speed_ms,0,blend_radius_m)
    |   movel([0.129970, -1.263701, -2.646341, -0.802347, 1.570796, 1.700766],accel_mss,speed_ms,0,blend_radius_m)
    |   movel([0.128563, -1.263661, -2.646363, -0.802365, 1.570796, 1.699359],accel_mss,speed_ms,0,blend_radius_m)
    |   # Splitting Linear movement in 16 (instruction 30: MoveL 25)
    |   movel([0.128563, -1.262171, -2.645660, -0.804557, 1.570796, 1.699359],accel_mss,speed_ms,0,blend_radius_m)
    |   movel([0.128563, -1.260687, -2.644956, -0.806746, 1.570796, 1.699359],accel_mss,speed_ms,0,blend_radius_m)
    |   movel([0.128563, -1.259208, -2.644250, -0.808930, 1.570796, 1.699359],accel_mss,speed_ms,0,blend_radius_m)
    |   movel([0.128563, -1.257735, -2.643543, -0.811111, 1.570796, 1.699359],accel_mss,speed_ms,0,blend_radius_m)
    |   movel([0.128563, -1.256267, -2.642835, -0.813287, 1.570796, 1.699359],accel_mss,speed_ms,0,blend_radius_m)
    |   movel([0.128563, -1.254804, -2.642125, -0.815460, 1.570796, 1.699359],accel_mss,speed_ms,0,blend_radius_m)
    |   movel([0.128563, -1.253346, -2.641414, -0.817629, 1.570796, 1.699359],accel_mss,speed_ms,0,blend_radius_m)
    |   movel([0.128563, -1.251894, -2.640701, -0.819794, 1.570796, 1.699359],accel_mss,speed_ms,0,blend_radius_m)
    |   movel([0.128563, -1.250447, -2.639987, -0.821956, 1.570796, 1.699359],accel_mss,speed_ms,0,blend_radius_m)
    |   movel([0.128563, -1.249005, -2.639271, -0.824113, 1.570796, 1.699359],accel_mss,speed_ms,0,blend_radius_m)
    |   movel([0.128563, -1.247568, -2.638554, -0.826266, 1.570796, 1.699359],accel_mss,speed_ms,0,blend_radius_m)
    |   movel([0.128563, -1.246137, -2.637836, -0.828416, 1.570796, 1.699359],accel_mss,speed_ms,0,blend_radius_m)
    |   movel([0.128563, -1.244711, -2.637116, -0.830562, 1.570796, 1.699359],accel_mss,speed_ms,0,blend_radius_m)
    |   movel([0.128563, -1.243289, -2.636395, -0.832704, 1.570796, 1.699359],accel_mss,speed_ms,0,blend_radius_m)
    |   movel([0.128563, -1.241874, -2.635673, -0.834842, 1.570796, 1.699359],accel_mss,speed_ms,0,blend_radius_m)
    |   movel([0.128563, -1.240463, -2.634949, -0.836977, 1.570796, 1.699359],accel_mss,speed_ms,0,blend_radius_m)
    |   # Splitting Linear movement in 8 (instruction 31: MoveL 26)
    |   movel([0.129970, -1.240504, -2.634928, -0.836958, 1.570796, 1.700766],accel_mss,speed_ms,0,blend_radius_m)
    |   movel([0.131376, -1.240546, -2.634905, -0.836938, 1.570796, 1.702172],accel_mss,speed_ms,0,blend_radius_m)
    |   movel([0.132780, -1.240591, -2.634881, -0.836917, 1.570796, 1.703577],accel_mss,speed_ms,0,blend_radius_m)
    |   movel([0.134184, -1.240638, -2.634856, -0.836895, 1.570796, 1.704980],accel_mss,speed_ms,0,blend_radius_m)
    |   movel([0.135586, -1.240688, -2.634830, -0.836872, 1.570796, 1.706382],accel_mss,speed_ms,0,blend_radius_m)
    |   movel([0.136987, -1.240739, -2.634802, -0.836847, 1.570796, 1.707784],accel_mss,speed_ms,0,blend_radius_m)
    |   movel([0.138387, -1.240793, -2.634774, -0.836822, 1.570796, 1.709184],accel_mss,speed_ms,0,blend_radius_m)
    |   movel([0.139786, -1.240849, -2.634744, -0.836796, 1.570796, 1.710582],accel_mss,speed_ms,0,blend_radius_m)
    |   # Splitting Linear movement in 16 (instruction 32: MoveL 27)
    |   movel([0.139786, -1.242259, -2.635467, -0.834662, 1.570796, 1.710582],accel_mss,speed_ms,0,blend_radius_m)
    |   movel([0.139786, -1.243675, -2.636189, -0.832524, 1.570796, 1.710582],accel_mss,speed_ms,0,blend_radius_m)
    |   movel([0.139786, -1.245096, -2.636910, -0.830383, 1.570796, 1.710582],accel_mss,speed_ms,0,blend_radius_m)
    |   movel([0.139786, -1.246522, -2.637630, -0.828238, 1.570796, 1.710582],accel_mss,speed_ms,0,blend_radius_m)
    |   movel([0.139786, -1.247953, -2.638348, -0.826088, 1.570796, 1.710582],accel_mss,speed_ms,0,blend_radius_m)
    |   movel([0.139786, -1.249389, -2.639064, -0.823935, 1.570796, 1.710582],accel_mss,speed_ms,0,blend_radius_m)
    |   movel([0.139786, -1.250831, -2.639779, -0.821778, 1.570796, 1.710582],accel_mss,speed_ms,0,blend_radius_m)
    |   movel([0.139786, -1.252278, -2.640493, -0.819618, 1.570796, 1.710582],accel_mss,speed_ms,0,blend_radius_m)
    |   movel([0.139786, -1.253730, -2.641206, -0.817453, 1.570796, 1.710582],accel_mss,speed_ms,0,blend_radius_m)
    |   movel([0.139786, -1.255187, -2.641917, -0.815285, 1.570796, 1.710582],accel_mss,speed_ms,0,blend_radius_m)
    |   movel([0.139786, -1.256650, -2.642626, -0.813113, 1.570796, 1.710582],accel_mss,speed_ms,0,blend_radius_m)
    |   movel([0.139786, -1.258118, -2.643335, -0.810936, 1.570796, 1.710582],accel_mss,speed_ms,0,blend_radius_m)
    |   movel([0.139786, -1.259591, -2.644041, -0.808756, 1.570796, 1.710582],accel_mss,speed_ms,0,blend_radius_m)
    |   movel([0.139786, -1.261070, -2.644747, -0.806573, 1.570796, 1.710582],accel_mss,speed_ms,0,blend_radius_m)
    |   movel([0.139786, -1.262553, -2.645451, -0.804385, 1.570796, 1.710582],accel_mss,speed_ms,0,blend_radius_m)
    |   movel([0.139786, -1.264042, -2.646153, -0.802193, 1.570796, 1.710582],accel_mss,speed_ms,0,blend_radius_m)
    |   # Splitting Linear movement in 8 (instruction 33: MoveL 28)
    |   movel([0.138231, -1.265014, -2.645619, -0.801756, 1.570796, 1.709027],accel_mss,speed_ms,0,blend_radius_m)
    |   movel([0.136677, -1.265986, -2.645083, -0.801320, 1.570796, 1.707474],accel_mss,speed_ms,0,blend_radius_m)
    |   movel([0.135127, -1.266957, -2.644546, -0.800886, 1.570796, 1.705923],accel_mss,speed_ms,0,blend_radius_m)
    |   movel([0.133578, -1.267928, -2.644009, -0.800453, 1.570796, 1.704374],accel_mss,speed_ms,0,blend_radius_m)
    |   movel([0.132032, -1.268898, -2.643470, -0.800021, 1.570796, 1.702828],accel_mss,speed_ms,0,blend_radius_m)
    |   movel([0.130488, -1.269869, -2.642930, -0.799590, 1.570796, 1.701284],accel_mss,speed_ms,0,blend_radius_m)
    |   movel([0.128946, -1.270838, -2.642390, -0.799161, 1.570796, 1.699743],accel_mss,speed_ms,0,blend_radius_m)
    |   movel([0.127407, -1.271808, -2.641848, -0.798733, 1.570796, 1.698204],accel_mss,speed_ms,0,blend_radius_m)
    |   # Splitting Linear movement in 16 (instruction 34: MoveL 29)
    |   movel([0.127407, -1.270325, -2.641151, -0.800912, 1.570796, 1.698204],accel_mss,speed_ms,0,blend_radius_m)
    |   movel([0.127407, -1.268848, -2.640453, -0.803088, 1.570796, 1.698204],accel_mss,speed_ms,0,blend_radius_m)
    |   movel([0.127407, -1.267376, -2.639753, -0.805260, 1.570796, 1.698204],accel_mss,speed_ms,0,blend_radius_m)
    |   movel([0.127407, -1.265909, -2.639052, -0.807429, 1.570796, 1.698204],accel_mss,speed_ms,0,blend_radius_m)
    |   movel([0.127407, -1.264447, -2.638349, -0.809593, 1.570796, 1.698204],accel_mss,speed_ms,0,blend_radius_m)
    |   movel([0.127407, -1.262990, -2.637645, -0.811754, 1.570796, 1.698204],accel_mss,speed_ms,0,blend_radius_m)
    |   movel([0.127407, -1.261539, -2.636939, -0.813911, 1.570796, 1.698204],accel_mss,speed_ms,0,blend_radius_m)
    |   movel([0.127407, -1.260092, -2.636232, -0.816064, 1.570796, 1.698204],accel_mss,speed_ms,0,blend_radius_m)
    |   movel([0.127407, -1.258651, -2.635524, -0.818214, 1.570796, 1.698204],accel_mss,speed_ms,0,blend_radius_m)
    |   movel([0.127407, -1.257215, -2.634814, -0.820360, 1.570796, 1.698204],accel_mss,speed_ms,0,blend_radius_m)
    |   movel([0.127407, -1.255784, -2.634103, -0.822502, 1.570796, 1.698204],accel_mss,speed_ms,0,blend_radius_m)
    |   movel([0.127407, -1.254358, -2.633391, -0.824640, 1.570796, 1.698204],accel_mss,speed_ms,0,blend_radius_m)
    |   movel([0.127407, -1.252938, -2.632677, -0.826775, 1.570796, 1.698204],accel_mss,speed_ms,0,blend_radius_m)
    |   movel([0.127407, -1.251522, -2.631961, -0.828906, 1.570796, 1.698204],accel_mss,speed_ms,0,blend_radius_m)
    |   movel([0.127407, -1.250112, -2.631245, -0.831033, 1.570796, 1.698204],accel_mss,speed_ms,0,blend_radius_m)
    |   movel([0.127407, -1.248706, -2.630527, -0.833156, 1.570796, 1.698204],accel_mss,speed_ms,0,blend_radius_m)
    |   # Splitting Linear movement in 6 (instruction 35: MoveL 30)
    |   movel([0.128215, -1.247387, -2.631240, -0.833762, 1.570796, 1.699011],accel_mss,speed_ms,0,blend_radius_m)
    |   movel([0.129025, -1.246065, -2.631952, -0.834372, 1.570796, 1.699822],accel_mss,speed_ms,0,blend_radius_m)
    |   movel([0.129837, -1.244740, -2.632664, -0.834984, 1.570796, 1.700634],accel_mss,speed_ms,0,blend_radius_m)
    |   movel([0.130652, -1.243413, -2.633376, -0.835600, 1.570796, 1.701448],accel_mss,speed_ms,0,blend_radius_m)
    |   movel([0.131468, -1.242082, -2.634087, -0.836220, 1.570796, 1.702265],accel_mss,speed_ms,0,blend_radius_m)
    |   movel([0.132287, -1.240749, -2.634797, -0.836843, 1.570796, 1.703083],accel_mss,speed_ms,0,blend_radius_m)
    |   # Splitting Linear movement in 16 (instruction 36: MoveL 31)
    |   movel([0.132287, -1.242160, -2.635521, -0.834709, 1.570796, 1.703083],accel_mss,speed_ms,0,blend_radius_m)
    |   movel([0.132287, -1.243575, -2.636243, -0.832571, 1.570796, 1.703083],accel_mss,speed_ms,0,blend_radius_m)
    |   movel([0.132287, -1.244996, -2.636964, -0.830429, 1.570796, 1.703083],accel_mss,speed_ms,0,blend_radius_m)
    |   movel([0.132287, -1.246422, -2.637683, -0.828284, 1.570796, 1.703083],accel_mss,speed_ms,0,blend_radius_m)
    |   movel([0.132287, -1.247853, -2.638401, -0.826134, 1.570796, 1.703083],accel_mss,speed_ms,0,blend_radius_m)
    |   movel([0.132287, -1.249290, -2.639118, -0.823981, 1.570796, 1.703083],accel_mss,speed_ms,0,blend_radius_m)
    |   movel([0.132287, -1.250732, -2.639833, -0.821824, 1.570796, 1.703083],accel_mss,speed_ms,0,blend_radius_m)
    |   movel([0.132287, -1.252178, -2.640547, -0.819663, 1.570796, 1.703083],accel_mss,speed_ms,0,blend_radius_m)
    |   movel([0.132287, -1.253631, -2.641260, -0.817499, 1.570796, 1.703083],accel_mss,speed_ms,0,blend_radius_m)
    |   movel([0.132287, -1.255088, -2.641971, -0.815330, 1.570796, 1.703083],accel_mss,speed_ms,0,blend_radius_m)
    |   movel([0.132287, -1.256551, -2.642680, -0.813158, 1.570796, 1.703083],accel_mss,speed_ms,0,blend_radius_m)
    |   movel([0.132287, -1.258019, -2.643389, -0.810982, 1.570796, 1.703083],accel_mss,speed_ms,0,blend_radius_m)
    |   movel([0.132287, -1.259492, -2.644096, -0.808801, 1.570796, 1.703083],accel_mss,speed_ms,0,blend_radius_m)
    |   movel([0.132287, -1.260971, -2.644801, -0.806617, 1.570796, 1.703083],accel_mss,speed_ms,0,blend_radius_m)
    |   movel([0.132287, -1.262454, -2.645505, -0.804429, 1.570796, 1.703083],accel_mss,speed_ms,0,blend_radius_m)
    |   movel([0.132287, -1.263944, -2.646208, -0.802238, 1.570796, 1.703083],accel_mss,speed_ms,0,blend_radius_m)
    |   movel([0.131542, -1.269052, -2.643385, -0.799952, 1.570796, 1.702338],accel_mss,speed_ms,0,blend_radius_m)
    |   # Splitting Linear movement in 16 (instruction 38: MoveL 33)
    |   movel([0.131542, -1.267567, -2.642686, -0.802136, 1.570796, 1.702338],accel_mss,speed_ms,0,blend_radius_m)
    |   movel([0.131542, -1.266088, -2.641985, -0.804316, 1.570796, 1.702338],accel_mss,speed_ms,0,blend_radius_m)
    |   movel([0.131542, -1.264613, -2.641283, -0.806493, 1.570796, 1.702338],accel_mss,speed_ms,0,blend_radius_m)
    |   movel([0.131542, -1.263144, -2.640580, -0.808665, 1.570796, 1.702338],accel_mss,speed_ms,0,blend_radius_m)
    |   movel([0.131542, -1.261680, -2.639875, -0.810834, 1.570796, 1.702338],accel_mss,speed_ms,0,blend_radius_m)
    |   movel([0.131542, -1.260221, -2.639169, -0.812999, 1.570796, 1.702338],accel_mss,speed_ms,0,blend_radius_m)
    |   movel([0.131542, -1.258767, -2.638462, -0.815160, 1.570796, 1.702338],accel_mss,speed_ms,0,blend_radius_m)
    |   movel([0.131542, -1.257319, -2.637753, -0.817317, 1.570796, 1.702338],accel_mss,speed_ms,0,blend_radius_m)
    |   movel([0.131542, -1.255876, -2.637043, -0.819471, 1.570796, 1.702338],accel_mss,speed_ms,0,blend_radius_m)
    |   movel([0.131542, -1.254438, -2.636331, -0.821620, 1.570796, 1.702338],accel_mss,speed_ms,0,blend_radius_m)
    |   movel([0.131542, -1.253005, -2.635618, -0.823766, 1.570796, 1.702338],accel_mss,speed_ms,0,blend_radius_m)
    |   movel([0.131542, -1.251577, -2.634903, -0.825909, 1.570796, 1.702338],accel_mss,speed_ms,0,blend_radius_m)
    |   movel([0.131542, -1.250154, -2.634188, -0.828047, 1.570796, 1.702338],accel_mss,speed_ms,0,blend_radius_m)
    |   movel([0.131542, -1.248737, -2.633470, -0.830182, 1.570796, 1.702338],accel_mss,speed_ms,0,blend_radius_m)
    |   movel([0.131542, -1.247325, -2.632752, -0.832313, 1.570796, 1.702338],accel_mss,speed_ms,0,blend_radius_m)
    |   movel([0.131542, -1.245917, -2.632032, -0.834440, 1.570796, 1.702338],accel_mss,speed_ms,0,blend_radius_m)
    |   # Splitting Linear movement in 6 (instruction 39: MoveL 34)
    |   movel([0.132749, -1.246189, -2.631885, -0.834314, 1.570796, 1.703546],accel_mss,speed_ms,0,blend_radius_m)
    |   movel([0.133955, -1.246463, -2.631738, -0.834188, 1.570796, 1.704752],accel_mss,speed_ms,0,blend_radius_m)
    |   movel([0.135160, -1.246739, -2.631589, -0.834061, 1.570796, 1.705956],accel_mss,speed_ms,0,blend_radius_m)
    |   movel([0.136363, -1.247016, -2.631440, -0.833933, 1.570796, 1.707159],accel_mss,speed_ms,0,blend_radius_m)
    |   movel([0.137564, -1.247295, -2.631289, -0.833804, 1.570796, 1.708361],accel_mss,speed_ms,0,blend_radius_m)
    |   movel([0.138764, -1.247576, -2.631138, -0.833675, 1.570796, 1.709561],accel_mss,speed_ms,0,blend_radius_m)
    |   # Splitting Linear movement in 16 (instruction 40: MoveL 35)
    |   movel([0.138764, -1.248982, -2.631856, -0.831550, 1.570796, 1.709561],accel_mss,speed_ms,0,blend_radius_m)
    |   movel([0.138764, -1.250394, -2.632574, -0.829421, 1.570796, 1.709561],accel_mss,speed_ms,0,blend_radius_m)
    |   movel([0.138764, -1.251810, -2.633290, -0.827289, 1.570796, 1.709561],accel_mss,speed_ms,0,blend_radius_m)
    |   movel([0.138764, -1.253232, -2.634005, -0.825153, 1.570796, 1.709561],accel_mss,speed_ms,0,blend_radius_m)
    |   movel([0.138764, -1.254658, -2.634718, -0.823013, 1.570796, 1.709561],accel_mss,speed_ms,0,blend_radius_m)
    |   movel([0.138764, -1.256090, -2.635430, -0.820869, 1.570796, 1.709561],accel_mss,speed_ms,0,blend_radius_m)
    |   movel([0.138764, -1.257527, -2.636140, -0.818722, 1.570796, 1.709561],accel_mss,speed_ms,0,blend_radius_m)
    |   movel([0.138764, -1.258969, -2.636849, -0.816571, 1.570796, 1.709561],accel_mss,speed_ms,0,blend_radius_m)
    |   movel([0.138764, -1.260416, -2.637557, -0.814416, 1.570796, 1.709561],accel_mss,speed_ms,0,blend_radius_m)
    |   movel([0.138764, -1.261868, -2.638264, -0.812257, 1.570796, 1.709561],accel_mss,speed_ms,0,blend_radius_m)
    |   movel([0.138764, -1.263326, -2.638968, -0.810095, 1.570796, 1.709561],accel_mss,speed_ms,0,blend_radius_m)
    |   movel([0.138764, -1.264789, -2.639672, -0.807928, 1.570796, 1.709561],accel_mss,speed_ms,0,blend_radius_m)
    |   movel([0.138764, -1.266256, -2.640374, -0.805758, 1.570796, 1.709561],accel_mss,speed_ms,0,blend_radius_m)
    |   movel([0.138764, -1.267730, -2.641075, -0.803585, 1.570796, 1.709561],accel_mss,speed_ms,0,blend_radius_m)
    |   movel([0.138764, -1.269208, -2.641774, -0.801407, 1.570796, 1.709561],accel_mss,speed_ms,0,blend_radius_m)
    |   movel([0.138764, -1.270692, -2.642472, -0.799226, 1.570796, 1.709561],accel_mss,speed_ms,0,blend_radius_m)
    |   # Splitting Linear movement in 6 (instruction 41: MoveL 36)
    |   movel([0.136810, -1.271293, -2.642136, -0.798960, 1.570796, 1.707606],accel_mss,speed_ms,0,blend_radius_m)
    |   movel([0.134856, -1.271896, -2.641799, -0.798694, 1.570796, 1.705653],accel_mss,speed_ms,0,blend_radius_m)
    |   movel([0.132903, -1.272502, -2.641460, -0.798427, 1.570796, 1.703700],accel_mss,speed_ms,0,blend_radius_m)
    |   movel([0.130952, -1.273110, -2.641119, -0.798160, 1.570796, 1.701748],accel_mss,speed_ms,0,blend_radius_m)
    |   movel([0.129001, -1.273720, -2.640777, -0.797892, 1.570796, 1.699797],accel_mss,speed_ms,0,blend_radius_m)
    |   movel([0.127050, -1.274333, -2.640433, -0.797624, 1.570796, 1.697847],accel_mss,speed_ms,0,blend_radius_m)
    |   # Splitting Linear movement in 16 (instruction 42: MoveL 37)
    |   movel([0.127050, -1.272852, -2.639737, -0.799800, 1.570796, 1.697847],accel_mss,speed_ms,0,blend_radius_m)
    |   movel([0.127050, -1.271377, -2.639041, -0.801972, 1.570796, 1.697847],accel_mss,speed_ms,0,blend_radius_m)
    |   movel([0.127050, -1.269907, -2.638343, -0.804140, 1.570796, 1.697847],accel_mss,speed_ms,0,blend_radius_m)
    |   movel([0.127050, -1.268442, -2.637643, -0.806304, 1.570796, 1.697847],accel_mss,speed_ms,0,blend_radius_m)
    |   movel([0.127050, -1.266982, -2.636942, -0.808465, 1.570796, 1.697847],accel_mss,speed_ms,0,blend_radius_m)
    |   movel([0.127050, -1.265527, -2.636240, -0.810622, 1.570796, 1.697847],accel_mss,speed_ms,0,blend_radius_m)
    |   movel([0.127050, -1.264078, -2.635536, -0.812775, 1.570796, 1.697847],accel_mss,speed_ms,0,blend_radius_m)
    |   movel([0.127050, -1.262633, -2.634831, -0.814925, 1.570796, 1.697847],accel_mss,speed_ms,0,blend_radius_m)
    |   movel([0.127050, -1.261194, -2.634124, -0.817071, 1.570796, 1.697847],accel_mss,speed_ms,0,blend_radius_m)
    |   movel([0.127050, -1.259760, -2.633416, -0.819213, 1.570796, 1.697847],accel_mss,speed_ms,0,blend_radius_m)
    |   movel([0.127050, -1.258330, -2.632707, -0.821351, 1.570796, 1.697847],accel_mss,speed_ms,0,blend_radius_m)
    |   movel([0.127050, -1.256906, -2.631996, -0.823486, 1.570796, 1.697847],accel_mss,speed_ms,0,blend_radius_m)
    |   movel([0.127050, -1.255488, -2.631284, -0.825617, 1.570796, 1.697847],accel_mss,speed_ms,0,blend_radius_m)
    |   movel([0.127050, -1.254074, -2.630571, -0.827745, 1.570796, 1.697847],accel_mss,speed_ms,0,blend_radius_m)
    |   movel([0.127050, -1.252665, -2.629856, -0.829868, 1.570796, 1.697847],accel_mss,speed_ms,0,blend_radius_m)
    |   movel([0.127050, -1.251261, -2.629140, -0.831988, 1.570796, 1.697847],accel_mss,speed_ms,0,blend_radius_m)
    |   # Splitting Linear movement in 6 (instruction 43: MoveL 38)
    |   movel([0.129001, -1.250641, -2.629477, -0.832271, 1.570796, 1.699797],accel_mss,speed_ms,0,blend_radius_m)
    |   movel([0.130952, -1.250023, -2.629813, -0.832553, 1.570796, 1.701748],accel_mss,speed_ms,0,blend_radius_m)
    |   movel([0.132903, -1.249408, -2.630146, -0.832835, 1.570796, 1.703700],accel_mss,speed_ms,0,blend_radius_m)
    |   movel([0.134856, -1.248795, -2.630479, -0.833115, 1.570796, 1.705653],accel_mss,speed_ms,0,blend_radius_m)
    |   movel([0.136810, -1.248184, -2.630809, -0.833396, 1.570796, 1.707606],accel_mss,speed_ms,0,blend_radius_m)
    |   movel([0.138764, -1.247576, -2.631138, -0.833675, 1.570796, 1.709561],accel_mss,speed_ms,0,blend_radius_m)
    |   # Splitting Linear movement in 16 (instruction 44: MoveL 39)
    |   movel([0.138764, -1.248982, -2.631856, -0.831550, 1.570796, 1.709561],accel_mss,speed_ms,0,blend_radius_m)
    |   movel([0.138764, -1.250394, -2.632574, -0.829421, 1.570796, 1.709561],accel_mss,speed_ms,0,blend_radius_m)
    |   movel([0.138764, -1.251810, -2.633290, -0.827289, 1.570796, 1.709561],accel_mss,speed_ms,0,blend_radius_m)
    |   movel([0.138764, -1.253232, -2.634005, -0.825153, 1.570796, 1.709561],accel_mss,speed_ms,0,blend_radius_m)
    |   movel([0.138764, -1.254658, -2.634718, -0.823013, 1.570796, 1.709561],accel_mss,speed_ms,0,blend_radius_m)
    |   movel([0.138764, -1.256090, -2.635430, -0.820869, 1.570796, 1.709561],accel_mss,speed_ms,0,blend_radius_m)
    |   movel([0.138764, -1.257527, -2.636140, -0.818722, 1.570796, 1.709561],accel_mss,speed_ms,0,blend_radius_m)
    |   movel([0.138764, -1.258969, -2.636849, -0.816571, 1.570796, 1.709561],accel_mss,speed_ms,0,blend_radius_m)
    |   movel([0.138764, -1.260416, -2.637557, -0.814416, 1.570796, 1.709561],accel_mss,speed_ms,0,blend_radius_m)
    |   movel([0.138764, -1.261868, -2.638264, -0.812257, 1.570796, 1.709561],accel_mss,speed_ms,0,blend_radius_m)
    |   movel([0.138764, -1.263326, -2.638968, -0.810095, 1.570796, 1.709561],accel_mss,speed_ms,0,blend_radius_m)
    |   movel([0.138764, -1.264789, -2.639672, -0.807928, 1.570796, 1.709561],accel_mss,speed_ms,0,blend_radius_m)
    |   movel([0.138764, -1.266256, -2.640374, -0.805758, 1.570796, 1.709561],accel_mss,speed_ms,0,blend_radius_m)
    |   movel([0.138764, -1.267730, -2.641075, -0.803585, 1.570796, 1.709561],accel_mss,speed_ms,0,blend_radius_m)
    |   movel([0.138764, -1.269208, -2.641774, -0.801407, 1.570796, 1.709561],accel_mss,speed_ms,0,blend_radius_m)
    |   movel([0.138764, -1.270692, -2.642472, -0.799226, 1.570796, 1.709561],accel_mss,speed_ms,0,blend_radius_m)
    |   movel([0.138066, -1.275254, -2.639914, -0.797221, 1.570796, 1.708862],accel_mss,speed_ms,0,blend_radius_m)
    |   movel([0.137280, -1.276937, -2.638964, -0.796488, 1.570796, 1.708076],accel_mss,speed_ms,0,blend_radius_m)
    |   movel([0.136649, -1.277609, -2.638584, -0.796197, 1.570796, 1.707445],accel_mss,speed_ms,0,blend_radius_m)
    |   movel([0.135466, -1.278449, -2.638107, -0.795833, 1.570796, 1.706262],accel_mss,speed_ms,0,blend_radius_m)
    |   movel([0.134358, -1.278787, -2.637915, -0.795687, 1.570796, 1.705154],accel_mss,speed_ms,0,blend_radius_m)
    |   movel([0.133325, -1.278625, -2.638007, -0.795757, 1.570796, 1.704122],accel_mss,speed_ms,0,blend_radius_m)
    |   movel([0.132845, -1.278293, -2.638195, -0.795900, 1.570796, 1.703642],accel_mss,speed_ms,0,blend_radius_m)
    |   movel([0.132513, -1.276957, -2.638952, -0.796480, 1.570796, 1.703309],accel_mss,speed_ms,0,blend_radius_m)
    |   movel([0.133182, -1.272415, -2.641509, -0.798465, 1.570796, 1.703979],accel_mss,speed_ms,0,blend_radius_m)
    |   # Splitting Linear movement in 16 (instruction 54: MoveL 49)
    |   movel([0.133182, -1.270933, -2.640812, -0.800644, 1.570796, 1.703979],accel_mss,speed_ms,0,blend_radius_m)
    |   movel([0.133182, -1.269456, -2.640114, -0.802819, 1.570796, 1.703979],accel_mss,speed_ms,0,blend_radius_m)
    |   movel([0.133182, -1.267984, -2.639415, -0.804990, 1.570796, 1.703979],accel_mss,speed_ms,0,blend_radius_m)
    |   movel([0.133182, -1.266518, -2.638714, -0.807158, 1.570796, 1.703979],accel_mss,speed_ms,0,blend_radius_m)
    |   movel([0.133182, -1.265056, -2.638011, -0.809321, 1.570796, 1.703979],accel_mss,speed_ms,0,blend_radius_m)
    |   movel([0.133182, -1.263600, -2.637308, -0.811481, 1.570796, 1.703979],accel_mss,speed_ms,0,blend_radius_m)
    |   movel([0.133182, -1.262149, -2.636603, -0.813637, 1.570796, 1.703979],accel_mss,speed_ms,0,blend_radius_m)
    |   movel([0.133182, -1.260703, -2.635896, -0.815790, 1.570796, 1.703979],accel_mss,speed_ms,0,blend_radius_m)
    |   movel([0.133182, -1.259262, -2.635188, -0.817938, 1.570796, 1.703979],accel_mss,speed_ms,0,blend_radius_m)
    |   movel([0.133182, -1.257827, -2.634479, -0.820083, 1.570796, 1.703979],accel_mss,speed_ms,0,blend_radius_m)
    |   movel([0.133182, -1.256396, -2.633768, -0.822225, 1.570796, 1.703979],accel_mss,speed_ms,0,blend_radius_m)
    |   movel([0.133182, -1.254971, -2.633056, -0.824362, 1.570796, 1.703979],accel_mss,speed_ms,0,blend_radius_m)
    |   movel([0.133182, -1.253551, -2.632343, -0.826496, 1.570796, 1.703979],accel_mss,speed_ms,0,blend_radius_m)
    |   movel([0.133182, -1.252135, -2.631628, -0.828626, 1.570796, 1.703979],accel_mss,speed_ms,0,blend_radius_m)
    |   movel([0.133182, -1.250725, -2.630912, -0.830752, 1.570796, 1.703979],accel_mss,speed_ms,0,blend_radius_m)
    |   movel([0.133182, -1.249320, -2.630194, -0.832875, 1.570796, 1.703979],accel_mss,speed_ms,0,blend_radius_m)
    |   movel([0.132661, -1.252899, -2.628247, -0.831244, 1.570796, 1.703458],accel_mss,speed_ms,0,blend_radius_m)
    |   # Splitting Linear movement in 16 (instruction 56: MoveL 51)
    |   movel([0.132661, -1.254301, -2.628962, -0.829126, 1.570796, 1.703458],accel_mss,speed_ms,0,blend_radius_m)
    |   movel([0.132661, -1.255709, -2.629675, -0.827005, 1.570796, 1.703458],accel_mss,speed_ms,0,blend_radius_m)
    |   movel([0.132661, -1.257122, -2.630388, -0.824879, 1.570796, 1.703458],accel_mss,speed_ms,0,blend_radius_m)
    |   movel([0.132661, -1.258540, -2.631099, -0.822751, 1.570796, 1.703458],accel_mss,speed_ms,0,blend_radius_m)
    |   movel([0.132661, -1.259962, -2.631808, -0.820618, 1.570796, 1.703458],accel_mss,speed_ms,0,blend_radius_m)
    |   movel([0.132661, -1.261390, -2.632516, -0.818482, 1.570796, 1.703458],accel_mss,speed_ms,0,blend_radius_m)
    |   movel([0.132661, -1.262823, -2.633223, -0.816342, 1.570796, 1.703458],accel_mss,speed_ms,0,blend_radius_m)
    |   movel([0.132661, -1.264261, -2.633929, -0.814199, 1.570796, 1.703458],accel_mss,speed_ms,0,blend_radius_m)
    |   movel([0.132661, -1.265705, -2.634633, -0.812052, 1.570796, 1.703458],accel_mss,speed_ms,0,blend_radius_m)
    |   movel([0.132661, -1.267153, -2.635335, -0.809901, 1.570796, 1.703458],accel_mss,speed_ms,0,blend_radius_m)
    |   movel([0.132661, -1.268606, -2.636037, -0.807746, 1.570796, 1.703458],accel_mss,speed_ms,0,blend_radius_m)
    |   movel([0.132661, -1.270065, -2.636736, -0.805588, 1.570796, 1.703458],accel_mss,speed_ms,0,blend_radius_m)
    |   movel([0.132661, -1.271529, -2.637435, -0.803426, 1.570796, 1.703458],accel_mss,speed_ms,0,blend_radius_m)
    |   movel([0.132661, -1.272997, -2.638132, -0.801260, 1.570796, 1.703458],accel_mss,speed_ms,0,blend_radius_m)
    |   movel([0.132661, -1.274471, -2.638827, -0.799091, 1.570796, 1.703458],accel_mss,speed_ms,0,blend_radius_m)
    |   movel([0.132661, -1.275950, -2.639521, -0.796917, 1.570796, 1.703458],accel_mss,speed_ms,0,blend_radius_m)
    |   # Splitting Linear movement in 4 (instruction 57: MoveL 52)
    |   movel([0.131006, -1.277303, -2.638757, -0.796329, 1.570796, 1.701802],accel_mss,speed_ms,0,blend_radius_m)
    |   movel([0.129354, -1.278654, -2.637991, -0.795744, 1.570796, 1.700150],accel_mss,speed_ms,0,blend_radius_m)
    |   movel([0.127706, -1.280002, -2.637224, -0.795163, 1.570796, 1.698502],accel_mss,speed_ms,0,blend_radius_m)
    |   movel([0.126062, -1.281349, -2.636456, -0.794584, 1.570796, 1.696859],accel_mss,speed_ms,0,blend_radius_m)
    |   # Splitting Linear movement in 16 (instruction 58: MoveL 53)
    |   movel([0.126062, -1.279874, -2.635766, -0.796748, 1.570796, 1.696859],accel_mss,speed_ms,0,blend_radius_m)
    |   movel([0.126062, -1.278405, -2.635074, -0.798910, 1.570796, 1.696859],accel_mss,speed_ms,0,blend_radius_m)
    |   movel([0.126062, -1.276941, -2.634381, -0.801067, 1.570796, 1.696859],accel_mss,speed_ms,0,blend_radius_m)
    |   movel([0.126062, -1.275482, -2.633687, -0.803221, 1.570796, 1.696859],accel_mss,speed_ms,0,blend_radius_m)
    |   movel([0.126062, -1.274027, -2.632991, -0.805371, 1.570796, 1.696859],accel_mss,speed_ms,0,blend_radius_m)
    |   movel([0.126062, -1.272578, -2.632294, -0.807517, 1.570796, 1.696859],accel_mss,speed_ms,0,blend_radius_m)
    |   movel([0.126062, -1.271134, -2.631595, -0.809660, 1.570796, 1.696859],accel_mss,speed_ms,0,blend_radius_m)
    |   movel([0.126062, -1.269695, -2.630895, -0.811799, 1.570796, 1.696859],accel_mss,speed_ms,0,blend_radius_m)
    |   movel([0.126062, -1.268261, -2.630193, -0.813935, 1.570796, 1.696859],accel_mss,speed_ms,0,blend_radius_m)
    |   movel([0.126062, -1.266832, -2.629490, -0.816067, 1.570796, 1.696859],accel_mss,speed_ms,0,blend_radius_m)
    |   movel([0.126062, -1.265409, -2.628786, -0.818195, 1.570796, 1.696859],accel_mss,speed_ms,0,blend_radius_m)
    |   movel([0.126062, -1.263990, -2.628080, -0.820320, 1.570796, 1.696859],accel_mss,speed_ms,0,blend_radius_m)
    |   movel([0.126062, -1.262576, -2.627373, -0.822441, 1.570796, 1.696859],accel_mss,speed_ms,0,blend_radius_m)
    |   movel([0.126062, -1.261167, -2.626664, -0.824558, 1.570796, 1.696859],accel_mss,speed_ms,0,blend_radius_m)
    |   movel([0.126062, -1.259763, -2.625954, -0.826672, 1.570796, 1.696859],accel_mss,speed_ms,0,blend_radius_m)
    |   movel([0.126062, -1.258364, -2.625243, -0.828782, 1.570796, 1.696859],accel_mss,speed_ms,0,blend_radius_m)
    |   # Splitting Linear movement in 8 (instruction 59: MoveL 54)
    |   movel([0.126982, -1.259340, -2.624702, -0.828346, 1.570796, 1.697779],accel_mss,speed_ms,0,blend_radius_m)
    |   movel([0.127900, -1.260317, -2.624161, -0.827911, 1.570796, 1.698696],accel_mss,speed_ms,0,blend_radius_m)
    |   movel([0.128815, -1.261294, -2.623617, -0.827477, 1.570796, 1.699611],accel_mss,speed_ms,0,blend_radius_m)
    |   movel([0.129727, -1.262272, -2.623073, -0.827044, 1.570796, 1.700524],accel_mss,speed_ms,0,blend_radius_m)
    |   movel([0.130637, -1.263250, -2.622527, -0.826612, 1.570796, 1.701434],accel_mss,speed_ms,0,blend_radius_m)
    |   movel([0.131545, -1.264229, -2.621980, -0.826181, 1.570796, 1.702341],accel_mss,speed_ms,0,blend_radius_m)
    |   movel([0.132450, -1.265208, -2.621431, -0.825751, 1.570796, 1.703246],accel_mss,speed_ms,0,blend_radius_m)
    |   movel([0.133352, -1.266187, -2.620881, -0.825321, 1.570796, 1.704149],accel_mss,speed_ms,0,blend_radius_m)
    |   # Splitting Linear movement in 16 (instruction 60: MoveL 55)
    |   movel([0.133352, -1.267580, -2.621587, -0.823222, 1.570796, 1.704149],accel_mss,speed_ms,0,blend_radius_m)
    |   movel([0.133352, -1.268979, -2.622291, -0.821119, 1.570796, 1.704149],accel_mss,speed_ms,0,blend_radius_m)
    |   movel([0.133352, -1.270382, -2.622994, -0.819013, 1.570796, 1.704149],accel_mss,speed_ms,0,blend_radius_m)
    |   movel([0.133352, -1.271790, -2.623696, -0.816903, 1.570796, 1.704149],accel_mss,speed_ms,0,blend_radius_m)
    |   movel([0.133352, -1.273203, -2.624396, -0.814789, 1.570796, 1.704149],accel_mss,speed_ms,0,blend_radius_m)
    |   movel([0.133352, -1.274621, -2.625095, -0.812672, 1.570796, 1.704149],accel_mss,speed_ms,0,blend_radius_m)
    |   movel([0.133352, -1.276044, -2.625793, -0.810552, 1.570796, 1.704149],accel_mss,speed_ms,0,blend_radius_m)
    |   movel([0.133352, -1.277472, -2.626489, -0.808428, 1.570796, 1.704149],accel_mss,speed_ms,0,blend_radius_m)
    |   movel([0.133352, -1.278905, -2.627184, -0.806300, 1.570796, 1.704149],accel_mss,speed_ms,0,blend_radius_m)
    |   movel([0.133352, -1.280343, -2.627877, -0.804169, 1.570796, 1.704149],accel_mss,speed_ms,0,blend_radius_m)
    |   movel([0.133352, -1.281785, -2.628569, -0.802035, 1.570796, 1.704149],accel_mss,speed_ms,0,blend_radius_m)
    |   movel([0.133352, -1.283233, -2.629259, -0.799897, 1.570796, 1.704149],accel_mss,speed_ms,0,blend_radius_m)
    |   movel([0.133352, -1.284686, -2.629948, -0.797755, 1.570796, 1.704149],accel_mss,speed_ms,0,blend_radius_m)
    |   movel([0.133352, -1.286143, -2.630636, -0.795610, 1.570796, 1.704149],accel_mss,speed_ms,0,blend_radius_m)
    |   movel([0.133352, -1.287606, -2.631322, -0.793461, 1.570796, 1.704149],accel_mss,speed_ms,0,blend_radius_m)
    |   movel([0.133352, -1.289074, -2.632007, -0.791309, 1.570796, 1.704149],accel_mss,speed_ms,0,blend_radius_m)
    |   movel([0.134520, -1.288250, -2.632485, -0.791654, 1.570796, 1.705317],accel_mss,speed_ms,0,blend_radius_m)
    |   movel([0.135765, -1.286931, -2.633249, -0.792209, 1.570796, 1.706562],accel_mss,speed_ms,0,blend_radius_m)
    |   movel([0.136464, -1.285774, -2.633917, -0.792698, 1.570796, 1.707260],accel_mss,speed_ms,0,blend_radius_m)
    |   movel([0.136766, -1.283784, -2.635062, -0.793543, 1.570796, 1.707562],accel_mss,speed_ms,0,blend_radius_m)
    |   movel([0.136367, -1.282952, -2.635539, -0.793898, 1.570796, 1.707163],accel_mss,speed_ms,0,blend_radius_m)
    |   movel([0.135416, -1.282287, -2.635920, -0.794182, 1.570796, 1.706212],accel_mss,speed_ms,0,blend_radius_m)
    |   movel([0.134388, -1.282122, -2.636014, -0.794252, 1.570796, 1.705184],accel_mss,speed_ms,0,blend_radius_m)
    |   movel([0.132808, -1.282127, -2.636011, -0.794250, 1.570796, 1.703604],accel_mss,speed_ms,0,blend_radius_m)
    |   movel([0.130051, -1.282972, -2.635528, -0.793889, 1.570796, 1.700847],accel_mss,speed_ms,0,blend_radius_m)
    |   movel([0.128326, -1.283978, -2.634951, -0.793461, 1.570796, 1.699123],accel_mss,speed_ms,0,blend_radius_m)
    |   movel([0.127155, -1.284813, -2.634470, -0.793106, 1.570796, 1.697951],accel_mss,speed_ms,0,blend_radius_m)
    |   movel([0.125915, -1.286144, -2.633703, -0.792542, 1.570796, 1.696712],accel_mss,speed_ms,0,blend_radius_m)
    |   movel([0.125228, -1.287302, -2.633034, -0.792053, 1.570796, 1.696024],accel_mss,speed_ms,0,blend_radius_m)
    |   movel([0.124952, -1.289274, -2.631890, -0.791225, 1.570796, 1.695748],accel_mss,speed_ms,0,blend_radius_m)
    |   movel([0.125361, -1.290090, -2.631416, -0.790883, 1.570796, 1.696158],accel_mss,speed_ms,0,blend_radius_m)
    |   movel([0.126317, -1.290737, -2.631038, -0.790613, 1.570796, 1.697113],accel_mss,speed_ms,0,blend_radius_m)
    |   movel([0.127339, -1.290895, -2.630947, -0.790547, 1.570796, 1.698136],accel_mss,speed_ms,0,blend_radius_m)
    |   # Splitting Linear movement in 16 (instruction 78: MoveL 73)
    |   movel([0.127339, -1.289429, -2.630263, -0.792697, 1.570796, 1.698136],accel_mss,speed_ms,0,blend_radius_m)
    |   movel([0.127339, -1.287968, -2.629578, -0.794843, 1.570796, 1.698136],accel_mss,speed_ms,0,blend_radius_m)
    |   movel([0.127339, -1.286512, -2.628892, -0.796985, 1.570796, 1.698136],accel_mss,speed_ms,0,blend_radius_m)
    |   movel([0.127339, -1.285061, -2.628204, -0.799124, 1.570796, 1.698136],accel_mss,speed_ms,0,blend_radius_m)
    |   movel([0.127339, -1.283615, -2.627515, -0.801259, 1.570796, 1.698136],accel_mss,speed_ms,0,blend_radius_m)
    |   movel([0.127339, -1.282174, -2.626824, -0.803391, 1.570796, 1.698136],accel_mss,speed_ms,0,blend_radius_m)
    |   movel([0.127339, -1.280737, -2.626132, -0.805519, 1.570796, 1.698136],accel_mss,speed_ms,0,blend_radius_m)
    |   movel([0.127339, -1.279306, -2.625439, -0.807644, 1.570796, 1.698136],accel_mss,speed_ms,0,blend_radius_m)
    |   movel([0.127339, -1.277880, -2.624744, -0.809765, 1.570796, 1.698136],accel_mss,speed_ms,0,blend_radius_m)
    |   movel([0.127339, -1.276458, -2.624048, -0.811883, 1.570796, 1.698136],accel_mss,speed_ms,0,blend_radius_m)
    |   movel([0.127339, -1.275042, -2.623350, -0.813997, 1.570796, 1.698136],accel_mss,speed_ms,0,blend_radius_m)
    |   movel([0.127339, -1.273630, -2.622651, -0.816108, 1.570796, 1.698136],accel_mss,speed_ms,0,blend_radius_m)
    |   movel([0.127339, -1.272223, -2.621951, -0.818215, 1.570796, 1.698136],accel_mss,speed_ms,0,blend_radius_m)
    |   movel([0.127339, -1.270821, -2.621249, -0.820319, 1.570796, 1.698136],accel_mss,speed_ms,0,blend_radius_m)
    |   movel([0.127339, -1.269424, -2.620546, -0.822419, 1.570796, 1.698136],accel_mss,speed_ms,0,blend_radius_m)
    |   movel([0.127339, -1.268032, -2.619841, -0.824516, 1.570796, 1.698136],accel_mss,speed_ms,0,blend_radius_m)
    |   # Splitting Linear movement in 6 (instruction 79: MoveL 74)
    |   movel([0.128655, -1.268579, -2.619532, -0.824278, 1.570796, 1.699451],accel_mss,speed_ms,0,blend_radius_m)
    |   movel([0.129968, -1.269128, -2.619222, -0.824040, 1.570796, 1.700764],accel_mss,speed_ms,0,blend_radius_m)
    |   movel([0.131278, -1.269678, -2.618910, -0.823801, 1.570796, 1.702075],accel_mss,speed_ms,0,blend_radius_m)
    |   movel([0.132586, -1.270231, -2.618596, -0.823561, 1.570796, 1.703383],accel_mss,speed_ms,0,blend_radius_m)
    |   movel([0.133892, -1.270787, -2.618281, -0.823321, 1.570796, 1.704688],accel_mss,speed_ms,0,blend_radius_m)
    |   movel([0.135195, -1.271344, -2.617965, -0.823081, 1.570796, 1.705991],accel_mss,speed_ms,0,blend_radius_m)
    |   # Splitting Linear movement in 16 (instruction 80: MoveL 75)
    |   movel([0.135195, -1.272733, -2.618667, -0.820989, 1.570796, 1.705991],accel_mss,speed_ms,0,blend_radius_m)
    |   movel([0.135195, -1.274128, -2.619368, -0.818893, 1.570796, 1.705991],accel_mss,speed_ms,0,blend_radius_m)
    |   movel([0.135195, -1.275528, -2.620067, -0.816794, 1.570796, 1.705991],accel_mss,speed_ms,0,blend_radius_m)
    |   movel([0.135195, -1.276932, -2.620766, -0.814692, 1.570796, 1.705991],accel_mss,speed_ms,0,blend_radius_m)
    |   movel([0.135195, -1.278341, -2.621462, -0.812586, 1.570796, 1.705991],accel_mss,speed_ms,0,blend_radius_m)
    |   movel([0.135195, -1.279755, -2.622158, -0.810476, 1.570796, 1.705991],accel_mss,speed_ms,0,blend_radius_m)
    |   movel([0.135195, -1.281174, -2.622852, -0.808363, 1.570796, 1.705991],accel_mss,speed_ms,0,blend_radius_m)
    |   movel([0.135195, -1.282598, -2.623544, -0.806247, 1.570796, 1.705991],accel_mss,speed_ms,0,blend_radius_m)
    |   movel([0.135195, -1.284026, -2.624235, -0.804127, 1.570796, 1.705991],accel_mss,speed_ms,0,blend_radius_m)
    |   movel([0.135195, -1.285460, -2.624925, -0.802004, 1.570796, 1.705991],accel_mss,speed_ms,0,blend_radius_m)
    |   movel([0.135195, -1.286898, -2.625613, -0.799877, 1.570796, 1.705991],accel_mss,speed_ms,0,blend_radius_m)
    |   movel([0.135195, -1.288341, -2.626300, -0.797747, 1.570796, 1.705991],accel_mss,speed_ms,0,blend_radius_m)
    |   movel([0.135195, -1.289790, -2.626986, -0.795614, 1.570796, 1.705991],accel_mss,speed_ms,0,blend_radius_m)
    |   movel([0.135195, -1.291243, -2.627670, -0.793477, 1.570796, 1.705991],accel_mss,speed_ms,0,blend_radius_m)
    |   movel([0.135195, -1.292701, -2.628352, -0.791336, 1.570796, 1.705991],accel_mss,speed_ms,0,blend_radius_m)
    |   movel([0.135195, -1.294164, -2.629033, -0.789192, 1.570796, 1.705991],accel_mss,speed_ms,0,blend_radius_m)
    |   movel([0.134799, -1.293344, -2.629514, -0.789530, 1.570796, 1.705595],accel_mss,speed_ms,0,blend_radius_m)
    |   movel([0.133857, -1.292686, -2.629900, -0.789803, 1.570796, 1.704653],accel_mss,speed_ms,0,blend_radius_m)
    |   movel([0.132841, -1.292521, -2.629997, -0.789872, 1.570796, 1.703637],accel_mss,speed_ms,0,blend_radius_m)
    |   movel([0.131279, -1.292520, -2.629997, -0.789872, 1.570796, 1.702075],accel_mss,speed_ms,0,blend_radius_m)
    |   movel([0.128555, -1.293342, -2.629516, -0.789531, 1.570796, 1.699351],accel_mss,speed_ms,0,blend_radius_m)
    |   movel([0.126852, -1.294326, -2.628938, -0.789125, 1.570796, 1.697648],accel_mss,speed_ms,0,blend_radius_m)
    |   movel([0.125695, -1.295144, -2.628457, -0.788788, 1.570796, 1.696491],accel_mss,speed_ms,0,blend_radius_m)
    |   movel([0.124472, -1.296450, -2.627687, -0.788252, 1.570796, 1.695268],accel_mss,speed_ms,0,blend_radius_m)
    |   movel([0.123794, -1.297588, -2.627015, -0.787787, 1.570796, 1.694590],accel_mss,speed_ms,0,blend_radius_m)
    |   movel([0.123525, -1.299528, -2.625864, -0.786997, 1.570796, 1.694321],accel_mss,speed_ms,0,blend_radius_m)
    |   movel([0.123931, -1.300333, -2.625385, -0.786671, 1.570796, 1.694727],accel_mss,speed_ms,0,blend_radius_m)
    |   movel([0.124876, -1.300974, -2.625003, -0.786412, 1.570796, 1.695673],accel_mss,speed_ms,0,blend_radius_m)
    |   movel([0.125888, -1.301132, -2.624909, -0.786348, 1.570796, 1.696684],accel_mss,speed_ms,0,blend_radius_m)
    |   movel([0.127438, -1.301131, -2.624910, -0.786349, 1.570796, 1.698235],accel_mss,speed_ms,0,blend_radius_m)
    |   movel([0.130138, -1.300326, -2.625389, -0.786674, 1.570796, 1.700934],accel_mss,speed_ms,0,blend_radius_m)
    |   movel([0.131830, -1.299359, -2.625964, -0.787066, 1.570796, 1.702626],accel_mss,speed_ms,0,blend_radius_m)
    |   movel([0.132983, -1.298553, -2.626443, -0.787393, 1.570796, 1.703779],accel_mss,speed_ms,0,blend_radius_m)
    |   movel([0.134211, -1.297258, -2.627209, -0.787921, 1.570796, 1.705007],accel_mss,speed_ms,0,blend_radius_m)
    |   movel([0.134900, -1.296122, -2.627881, -0.788386, 1.570796, 1.705696],accel_mss,speed_ms,0,blend_radius_m)
    |   movel([0.135195, -1.294164, -2.629033, -0.789192, 1.570796, 1.705991],accel_mss,speed_ms,0,blend_radius_m)
    |   movel([0.135195, -1.294164, -2.629033, -0.789192, 1.570796, 1.705991],accel_mss,speed_ms,0,blend_radius_m)
    |   # Splitting Linear movement in 72 (instruction 102: MoveL 97)
    |   movel([0.135195, -1.292539, -2.628276, -0.791574, 1.570796, 1.705991],accel_mss,speed_ms,0,blend_radius_m)
    |   movel([0.135195, -1.290919, -2.627518, -0.793952, 1.570796, 1.705991],accel_mss,speed_ms,0,blend_radius_m)
    |   movel([0.135195, -1.289306, -2.626757, -0.796325, 1.570796, 1.705991],accel_mss,speed_ms,0,blend_radius_m)
    |   movel([0.135195, -1.287699, -2.625995, -0.798694, 1.570796, 1.705991],accel_mss,speed_ms,0,blend_radius_m)
    |   movel([0.135195, -1.286098, -2.625231, -0.801059, 1.570796, 1.705991],accel_mss,speed_ms,0,blend_radius_m)
    |   movel([0.135195, -1.284504, -2.624465, -0.803420, 1.570796, 1.705991],accel_mss,speed_ms,0,blend_radius_m)
    |   movel([0.135195, -1.282915, -2.623698, -0.805776, 1.570796, 1.705991],accel_mss,speed_ms,0,blend_radius_m)
    |   movel([0.135195, -1.281332, -2.622929, -0.808128, 1.570796, 1.705991],accel_mss,speed_ms,0,blend_radius_m)
    |   movel([0.135195, -1.279755, -2.622158, -0.810476, 1.570796, 1.705991],accel_mss,speed_ms,0,blend_radius_m)
    |   movel([0.135195, -1.278184, -2.621385, -0.812820, 1.570796, 1.705991],accel_mss,speed_ms,0,blend_radius_m)
    |   movel([0.135195, -1.276619, -2.620611, -0.815159, 1.570796, 1.705991],accel_mss,speed_ms,0,blend_radius_m)
    |   movel([0.135195, -1.275061, -2.619834, -0.817494, 1.570796, 1.705991],accel_mss,speed_ms,0,blend_radius_m)
    |   movel([0.135195, -1.273508, -2.619057, -0.819825, 1.570796, 1.705991],accel_mss,speed_ms,0,blend_radius_m)
    |   movel([0.135195, -1.271961, -2.618277, -0.822151, 1.570796, 1.705991],accel_mss,speed_ms,0,blend_radius_m)
    |   movel([0.135195, -1.270420, -2.617496, -0.824473, 1.570796, 1.705991],accel_mss,speed_ms,0,blend_radius_m)
    |   movel([0.135195, -1.268885, -2.616713, -0.826791, 1.570796, 1.705991],accel_mss,speed_ms,0,blend_radius_m)
    |   movel([0.135195, -1.267356, -2.615928, -0.829105, 1.570796, 1.705991],accel_mss,speed_ms,0,blend_radius_m)
    |   movel([0.135195, -1.265833, -2.615142, -0.831415, 1.570796, 1.705991],accel_mss,speed_ms,0,blend_radius_m)
    |   movel([0.135195, -1.264315, -2.614354, -0.833720, 1.570796, 1.705991],accel_mss,speed_ms,0,blend_radius_m)
    |   movel([0.135195, -1.262804, -2.613564, -0.836021, 1.570796, 1.705991],accel_mss,speed_ms,0,blend_radius_m)
    |   movel([0.135195, -1.261298, -2.612773, -0.838318, 1.570796, 1.705991],accel_mss,speed_ms,0,blend_radius_m)
    |   movel([0.135195, -1.259799, -2.611980, -0.840610, 1.570796, 1.705991],accel_mss,speed_ms,0,blend_radius_m)
    |   movel([0.135195, -1.258305, -2.611185, -0.842899, 1.570796, 1.705991],accel_mss,speed_ms,0,blend_radius_m)
    |   movel([0.135195, -1.256817, -2.610389, -0.845183, 1.570796, 1.705991],accel_mss,speed_ms,0,blend_radius_m)
    |   movel([0.135195, -1.255335, -2.609591, -0.847463, 1.570796, 1.705991],accel_mss,speed_ms,0,blend_radius_m)
    |   movel([0.135195, -1.253859, -2.608791, -0.849739, 1.570796, 1.705991],accel_mss,speed_ms,0,blend_radius_m)
    |   movel([0.135195, -1.252388, -2.607990, -0.852011, 1.570796, 1.705991],accel_mss,speed_ms,0,blend_radius_m)
    |   movel([0.135195, -1.250924, -2.607187, -0.854278, 1.570796, 1.705991],accel_mss,speed_ms,0,blend_radius_m)
    |   movel([0.135195, -1.249465, -2.606383, -0.856541, 1.570796, 1.705991],accel_mss,speed_ms,0,blend_radius_m)
    |   movel([0.135195, -1.248012, -2.605577, -0.858800, 1.570796, 1.705991],accel_mss,speed_ms,0,blend_radius_m)
    |   movel([0.135195, -1.246565, -2.604769, -0.861055, 1.570796, 1.705991],accel_mss,speed_ms,0,blend_radius_m)
    |   movel([0.135195, -1.245123, -2.603960, -0.863306, 1.570796, 1.705991],accel_mss,speed_ms,0,blend_radius_m)
    |   movel([0.135195, -1.243687, -2.603149, -0.865553, 1.570796, 1.705991],accel_mss,speed_ms,0,blend_radius_m)
    |   movel([0.135195, -1.242257, -2.602336, -0.867795, 1.570796, 1.705991],accel_mss,speed_ms,0,blend_radius_m)
    |   movel([0.135195, -1.240833, -2.601522, -0.870034, 1.570796, 1.705991],accel_mss,speed_ms,0,blend_radius_m)
    |   movel([0.135195, -1.239414, -2.600707, -0.872268, 1.570796, 1.705991],accel_mss,speed_ms,0,blend_radius_m)
    |   movel([0.135195, -1.238001, -2.599890, -0.874498, 1.570796, 1.705991],accel_mss,speed_ms,0,blend_radius_m)
    |   movel([0.135195, -1.236594, -2.599071, -0.876724, 1.570796, 1.705991],accel_mss,speed_ms,0,blend_radius_m)
    |   movel([0.135195, -1.235192, -2.598251, -0.878946, 1.570796, 1.705991],accel_mss,speed_ms,0,blend_radius_m)
    |   movel([0.135195, -1.233796, -2.597429, -0.881164, 1.570796, 1.705991],accel_mss,speed_ms,0,blend_radius_m)
    |   movel([0.135195, -1.232406, -2.596606, -0.883378, 1.570796, 1.705991],accel_mss,speed_ms,0,blend_radius_m)
    |   movel([0.135195, -1.231021, -2.595781, -0.885587, 1.570796, 1.705991],accel_mss,speed_ms,0,blend_radius_m)
    |   movel([0.135195, -1.229642, -2.594954, -0.887793, 1.570796, 1.705991],accel_mss,speed_ms,0,blend_radius_m)
    |   movel([0.135195, -1.228268, -2.594126, -0.889994, 1.570796, 1.705991],accel_mss,speed_ms,0,blend_radius_m)
    |   movel([0.135195, -1.226900, -2.593297, -0.892192, 1.570796, 1.705991],accel_mss,speed_ms,0,blend_radius_m)
    |   movel([0.135195, -1.225538, -2.592466, -0.894385, 1.570796, 1.705991],accel_mss,speed_ms,0,blend_radius_m)
    |   movel([0.135195, -1.224181, -2.591633, -0.896574, 1.570796, 1.705991],accel_mss,speed_ms,0,blend_radius_m)
    |   movel([0.135195, -1.222830, -2.590799, -0.898760, 1.570796, 1.705991],accel_mss,speed_ms,0,blend_radius_m)
    |   movel([0.135195, -1.221484, -2.589964, -0.900941, 1.570796, 1.705991],accel_mss,speed_ms,0,blend_radius_m)
    |   movel([0.135195, -1.220144, -2.589127, -0.903118, 1.570796, 1.705991],accel_mss,speed_ms,0,blend_radius_m)
    |   movel([0.135195, -1.218809, -2.588289, -0.905291, 1.570796, 1.705991],accel_mss,speed_ms,0,blend_radius_m)
    |   movel([0.135195, -1.217480, -2.587449, -0.907460, 1.570796, 1.705991],accel_mss,speed_ms,0,blend_radius_m)
    |   movel([0.135195, -1.216156, -2.586607, -0.909626, 1.570796, 1.705991],accel_mss,speed_ms,0,blend_radius_m)
    |   movel([0.135195, -1.214838, -2.585764, -0.911787, 1.570796, 1.705991],accel_mss,speed_ms,0,blend_radius_m)
    |   movel([0.135195, -1.213525, -2.584920, -0.913944, 1.570796, 1.705991],accel_mss,speed_ms,0,blend_radius_m)
    |   movel([0.135195, -1.212218, -2.584074, -0.916097, 1.570796, 1.705991],accel_mss,speed_ms,0,blend_radius_m)
    |   movel([0.135195, -1.210916, -2.583227, -0.918246, 1.570796, 1.705991],accel_mss,speed_ms,0,blend_radius_m)
    |   movel([0.135195, -1.209619, -2.582378, -0.920392, 1.570796, 1.705991],accel_mss,speed_ms,0,blend_radius_m)
    |   movel([0.135195, -1.208328, -2.581528, -0.922533, 1.570796, 1.705991],accel_mss,speed_ms,0,blend_radius_m)
    |   movel([0.135195, -1.207042, -2.580676, -0.924670, 1.570796, 1.705991],accel_mss,speed_ms,0,blend_radius_m)
    |   movel([0.135195, -1.205762, -2.579823, -0.926804, 1.570796, 1.705991],accel_mss,speed_ms,0,blend_radius_m)
    |   movel([0.135195, -1.204487, -2.578969, -0.928933, 1.570796, 1.705991],accel_mss,speed_ms,0,blend_radius_m)
    |   movel([0.135195, -1.203217, -2.578113, -0.931059, 1.570796, 1.705991],accel_mss,speed_ms,0,blend_radius_m)
    |   movel([0.135195, -1.201953, -2.577256, -0.933180, 1.570796, 1.705991],accel_mss,speed_ms,0,blend_radius_m)
    |   movel([0.135195, -1.200694, -2.576397, -0.935298, 1.570796, 1.705991],accel_mss,speed_ms,0,blend_radius_m)
    |   movel([0.135195, -1.199440, -2.575537, -0.937412, 1.570796, 1.705991],accel_mss,speed_ms,0,blend_radius_m)
    |   movel([0.135195, -1.198192, -2.574675, -0.939522, 1.570796, 1.705991],accel_mss,speed_ms,0,blend_radius_m)
    |   movel([0.135195, -1.196949, -2.573812, -0.941628, 1.570796, 1.705991],accel_mss,speed_ms,0,blend_radius_m)
    |   movel([0.135195, -1.195711, -2.572948, -0.943730, 1.570796, 1.705991],accel_mss,speed_ms,0,blend_radius_m)
    |   movel([0.135195, -1.194478, -2.572082, -0.945829, 1.570796, 1.705991],accel_mss,speed_ms,0,blend_radius_m)
    |   movel([0.135195, -1.193251, -2.571215, -0.947923, 1.570796, 1.705991],accel_mss,speed_ms,0,blend_radius_m)
    |   movel([0.135195, -1.192029, -2.570347, -0.950014, 1.570796, 1.705991],accel_mss,speed_ms,0,blend_radius_m)
    |   # End of main program
    | end
    | 
    | Machining2()
